Universal Robots URScript: golden_headless.script

# UR5 - Protocole etalement cosmetique
# Genere automatiquement par ur5_etalement.py
# IMPORTANT : calibrer ROBOT_X_ORIGIN, ROBOT_Y_ORIGIN, ROBOT_Z_SURFACE avant execution
#
# === RECETTE DE REPRODUCTION ===
# Ce bloc enonce ce qui a produit ce fichier. Il ne porte pas de date :
# une date rendrait l export non reproductible, et git la porte deja.
# cycles : 6
#   cycle 1 : type=circular waypoints=83    label=Cycle 1 - Circulaire (0deg)
#   cycle 2 : type=circular waypoints=83    label=Cycle 2 - Circulaire (90deg)
#   cycle 3 : type=circular waypoints=83    label=Cycle 3 - Circulaire (0deg)
#   cycle 4 : type=linear   waypoints=26    label=Cycle 4 - Rectiligne (0deg)
#   cycle 5 : type=linear   waypoints=26    label=Cycle 5 - Rectiligne (90deg)
#   cycle 6 : type=linear   waypoints=26    label=Cycle 6 - Rectiligne (0deg)
# empreinte des reglages : 44136fa
#
# === PINCE 2F-85 : AUCUN ACTIONNEMENT ===
# Ce programme n a pas de commande de pince. La 2F-85 est un support
# passif pour le doigt silicone ; seule sa longueur (TCP_GRIPPER_Z=145 mm)
# entre dans set_tcp(). Aucun rq_activate / rq_* / RS485 outil / set_payload.
# Erreur PolyScope "wait for activation completed" au chargement = URCap
# Robotiq Grippers de l INSTALLATION du robot (auto-activation BeforeStart),
# pas ce fichier. Corriger sur le robot : Installation > URCaps/Gripper >
# desactiver l auto-activation, ou retirer le URCap, ou charger sur une
# installation sans pince.
#

# --- Ancre de la zone d'etalement ---
global P_REF = p[-0.011, 0.6, 0.05, 3.14159, 0.0, 0.0]

# --- Vitesses (m/s) par phase ---
# Note : URSCRIPT_MAX_TCP_SPEED (limite PolyScope, 0.25 m/s) n'est pas
# emis ici ; il est applique par le controleur. La vitesse de transit
# est inlinee directement sur les movel de transit.
global URSCRIPT_CONTACT_V = 0.0500  #sym:URSCRIPT_CONTACT_V
global URSCRIPT_RECONTACT_V = 0.0100  #sym:URSCRIPT_RECONTACT_V
global V_CIRC = 0.0360  #sym:CIRC_SPEED
global V_RECT = 0.0800  #sym:LIN_SPEED

# --- Accelerations (m/s^2) par phase ---
global URSCRIPT_ACCEL = 0.8  #sym:URSCRIPT_ACCEL
global A_INIT = 1.2  #sym:A_INIT

# --- Facteurs multiplicateurs globaux ---
global SPEED_FACTOR = 1.0
global ACCEL_FACTOR = 1.0
global URSCRIPT_BLEND = 0.002  #sym:URSCRIPT_BLEND

# --- Sondage de surface : 1 point en Z (sondage 3 points DESACTIVE, voir bloc commente) ---
global PROBE_FORCE_THR    = 4.0
global PROBE_DESCENT_V    = 0.0040
global PROBE_ACCEL        = 0.05
global PROBE_MAX_TRAVEL   = 0.15
global NOMINAL_FRAME = p[-0.011000, 0.592930, 0.050004, 3.141576, 0.000000, 0.000000]
global MEAS_FRAME = p[-0.011000, 0.592930, 0.050004, 3.141576, 0.000000, 0.000000]
global contact_found = False
global contact_pose = p[0,0,0,0,0,0]

# --- Sondage Z (1 point) : trouve le plan de la plaque par contact force ---
# Depart = pose courante (operateur jogge le doigt juste au-dessus du
# plateau). Descente en -Z (base) jusqu au contact ; le Z touche devient
# la reference de TOUS les cycles 1 a 6 via MEAS_FRAME.
def probe_surface_z():
  textmsg(">>> Sondage Z : 1 point (recherche du plateau)")
  start_pose = get_actual_tcp_pose()
  zero_ftsensor()
  sleep(0.2)
  # CB3 (PolyScope 3.x) : descente surveillee dans le thread principal
  # (speedl non bloquant + lecture force + stopl). Pas de thread (stopl/
  # movel interdits dans un thread). get_tcp_force() lu en entier, norme
  # calculee a la main (pas de slice [0:3], absent du parser CB3).
  f_norm = 0.0
  travel = 0.0
  while f_norm <= PROBE_FORCE_THR and travel < PROBE_MAX_TRAVEL:
    speedl([0, 0, -PROBE_DESCENT_V, 0, 0, 0], PROBE_ACCEL, 0.05)
    F_tcp = get_tcp_force()
    f_norm = sqrt(F_tcp[0]*F_tcp[0] + F_tcp[1]*F_tcp[1] + F_tcp[2]*F_tcp[2])
    cur = get_actual_tcp_pose()
    travel = start_pose[2] - cur[2]
  end
  stopl(2.0)
  if f_norm <= PROBE_FORCE_THR:
    popup("Sondage Z echoue - aucun contact", "Rapprocher le doigt du plateau puis relancer", error=True)
    halt
  end
  touch = get_actual_tcp_pose()
  # Reference Z des cycles : repere nominal translate en Z jusqu au plan
  # touche. Orientation/XY restent nominaux (1 point ne mesure pas
  # l inclinaison -> rework futur). apply_correction decale chaque
  # waypoint du meme dz ; force_mode(MEAS_FRAME) regule les 6 N en Z.
  MEAS_FRAME = p[NOMINAL_FRAME[0], NOMINAL_FRAME[1], touch[2], NOMINAL_FRAME[3], NOMINAL_FRAME[4], NOMINAL_FRAME[5]]
  textmsg("Plateau detecte, Z (m) = ", touch[2])
end

def apply_correction(p_world):
  return pose_trans(MEAS_FRAME, pose_trans(pose_inv(NOMINAL_FRAME), p_world))
end

def cycle_1():
  # --- Cycle 1 - Circulaire (0deg) ---
  movel(apply_correction(p[-0.017788, 0.586142, 0.060004, 3.141576, 0.000000, 0.000000]), a=URSCRIPT_ACCEL*ACCEL_FACTOR, v=0.2500*SPEED_FACTOR)
  sleep(0.2)
  zero_ftsensor()
  sleep(0.2)
  force_mode(MEAS_FRAME, [0, 0, 1, 0, 0, 0], [0, 0, -6.0, 0, 0, 0], 2, [0.008, 0.008, 0.04, 0.35, 0.35, 0.35])
  movel(apply_correction(p[-0.017788, 0.586142, 0.045004, 3.141576, 0.000000, 0.000000]), a=URSCRIPT_ACCEL*ACCEL_FACTOR, v=URSCRIPT_RECONTACT_V*SPEED_FACTOR)
  movel(apply_correction(p[-0.017788, 0.586142, 0.050004, 3.141576, 0.000000, 0.000000]), a=URSCRIPT_ACCEL*ACCEL_FACTOR, v=V_CIRC*SPEED_FACTOR, r=URSCRIPT_BLEND)
  movel(apply_correction(p[-0.005291, 0.586502, 0.050004, 3.141576, 0.000000, 0.000000]), a=URSCRIPT_ACCEL*ACCEL_FACTOR, v=V_CIRC*SPEED_FACTOR, r=URSCRIPT_BLEND)
  movel(apply_correction(p[-0.008415, 0.596171, 0.050004, 3.141576, 0.000000, 0.000000]), a=URSCRIPT_ACCEL*ACCEL_FACTOR, v=V_CIRC*SPEED_FACTOR, r=URSCRIPT_BLEND)
  movel(apply_correction(p[-0.016727, 0.588412, 0.050004, 3.141576, 0.000000, 0.000000]), a=URSCRIPT_ACCEL*ACCEL_FACTOR, v=V_CIRC*SPEED_FACTOR, r=URSCRIPT_BLEND)
  movel(apply_correction(p[-0.006870, 0.579901, 0.050004, 3.141576, 0.000000, 0.000000]), a=URSCRIPT_ACCEL*ACCEL_FACTOR, v=V_CIRC*SPEED_FACTOR, r=URSCRIPT_BLEND)
  movel(apply_correction(p[-0.000746, 0.589189, 0.050004, 3.141576, 0.000000, 0.000000]), a=URSCRIPT_ACCEL*ACCEL_FACTOR, v=V_CIRC*SPEED_FACTOR, r=URSCRIPT_BLEND)
  movel(apply_correction(p[-0.010687, 0.590761, 0.050004, 3.141576, 0.000000, 0.000000]), a=URSCRIPT_ACCEL*ACCEL_FACTOR, v=V_CIRC*SPEED_FACTOR, r=URSCRIPT_BLEND)
  movel(apply_correction(p[-0.009818, 0.578226, 0.050004, 3.141576, 0.000000, 0.000000]), a=URSCRIPT_ACCEL*ACCEL_FACTOR, v=V_CIRC*SPEED_FACTOR, r=URSCRIPT_BLEND)
  movel(apply_correction(p[0.002437, 0.579691, 0.050004, 3.141576, 0.000000, 0.000000]), a=URSCRIPT_ACCEL*ACCEL_FACTOR, v=V_CIRC*SPEED_FACTOR, r=URSCRIPT_BLEND)
  movel(apply_correction(p[-0.001599, 0.588917, 0.050004, 3.141576, 0.000000, 0.000000]), a=URSCRIPT_ACCEL*ACCEL_FACTOR, v=V_CIRC*SPEED_FACTOR, r=URSCRIPT_BLEND)
  movel(apply_correction(p[-0.009333, 0.580482, 0.050004, 3.141576, 0.000000, 0.000000]), a=URSCRIPT_ACCEL*ACCEL_FACTOR, v=V_CIRC*SPEED_FACTOR, r=URSCRIPT_BLEND)
  movel(apply_correction(p[0.000969, 0.572620, 0.050004, 3.141576, 0.000000, 0.000000]), a=URSCRIPT_ACCEL*ACCEL_FACTOR, v=V_CIRC*SPEED_FACTOR, r=URSCRIPT_BLEND)
  movel(apply_correction(p[0.006458, 0.582148, 0.050004, 3.141576, 0.000000, 0.000000]), a=URSCRIPT_ACCEL*ACCEL_FACTOR, v=V_CIRC*SPEED_FACTOR, r=URSCRIPT_BLEND)
  movel(apply_correction(p[-0.003817, 0.582897, 0.050004, 3.141576, 0.000000, 0.000000]), a=URSCRIPT_ACCEL*ACCEL_FACTOR, v=V_CIRC*SPEED_FACTOR, r=URSCRIPT_BLEND)
  movel(apply_correction(p[-0.001841, 0.570398, 0.050004, 3.141576, 0.000000, 0.000000]), a=URSCRIPT_ACCEL*ACCEL_FACTOR, v=V_CIRC*SPEED_FACTOR, r=URSCRIPT_BLEND)
  movel(apply_correction(p[0.010119, 0.572931, 0.050004, 3.141576, 0.000000, 0.000000]), a=URSCRIPT_ACCEL*ACCEL_FACTOR, v=V_CIRC*SPEED_FACTOR, r=URSCRIPT_BLEND)
  movel(apply_correction(p[0.005116, 0.581618, 0.050004, 3.141576, 0.000000, 0.000000]), a=URSCRIPT_ACCEL*ACCEL_FACTOR, v=V_CIRC*SPEED_FACTOR, r=URSCRIPT_BLEND)
  movel(apply_correction(p[-0.001866, 0.572369, 0.050004, 3.141576, 0.000000, 0.000000]), a=URSCRIPT_ACCEL*ACCEL_FACTOR, v=V_CIRC*SPEED_FACTOR, r=URSCRIPT_BLEND)
  movel(apply_correction(p[0.009049, 0.565429, 0.050004, 3.141576, 0.000000, 0.000000]), a=URSCRIPT_ACCEL*ACCEL_FACTOR, v=V_CIRC*SPEED_FACTOR, r=URSCRIPT_BLEND)
  movel(apply_correction(p[0.013497, 0.575336, 0.050004, 3.141576, 0.000000, 0.000000]), a=URSCRIPT_ACCEL*ACCEL_FACTOR, v=V_CIRC*SPEED_FACTOR, r=URSCRIPT_BLEND)
  movel(apply_correction(p[0.003100, 0.574984, 0.050004, 3.141576, 0.000000, 0.000000]), a=URSCRIPT_ACCEL*ACCEL_FACTOR, v=V_CIRC*SPEED_FACTOR, r=URSCRIPT_BLEND)
  movel(apply_correction(p[0.006175, 0.562627, 0.050005, 3.141576, 0.000000, 0.000000]), a=URSCRIPT_ACCEL*ACCEL_FACTOR, v=V_CIRC*SPEED_FACTOR, r=URSCRIPT_BLEND)
  movel(apply_correction(p[0.011479, 0.556739, 0.050005, 3.141576, 0.000000, 0.000000]), a=URSCRIPT_ACCEL*ACCEL_FACTOR, v=V_CIRC*SPEED_FACTOR, r=URSCRIPT_BLEND)
  movel(apply_correction(p[0.012647, 0.563823, 0.050005, 3.141576, 0.000000, 0.000000]), a=URSCRIPT_ACCEL*ACCEL_FACTOR, v=V_CIRC*SPEED_FACTOR, r=URSCRIPT_BLEND)
  movel(apply_correction(p[-0.002304, 0.566873, 0.050004, 3.141576, 0.000000, 0.000000]), a=URSCRIPT_ACCEL*ACCEL_FACTOR, v=V_CIRC*SPEED_FACTOR, r=URSCRIPT_BLEND)
  movel(apply_correction(p[-0.004889, 0.556556, 0.050005, 3.141576, 0.000000, 0.000000]), a=URSCRIPT_ACCEL*ACCEL_FACTOR, v=V_CIRC*SPEED_FACTOR, r=URSCRIPT_BLEND)
  movel(apply_correction(p[0.005466, 0.558816, 0.050005, 3.141576, 0.000000, 0.000000]), a=URSCRIPT_ACCEL*ACCEL_FACTOR, v=V_CIRC*SPEED_FACTOR, r=URSCRIPT_BLEND)
  movel(apply_correction(p[0.000547, 0.570683, 0.050004, 3.141576, 0.000000, 0.000000]), a=URSCRIPT_ACCEL*ACCEL_FACTOR, v=V_CIRC*SPEED_FACTOR, r=URSCRIPT_BLEND)
  movel(apply_correction(p[-0.010103, 0.565440, 0.050004, 3.141576, 0.000000, 0.000000]), a=URSCRIPT_ACCEL*ACCEL_FACTOR, v=V_CIRC*SPEED_FACTOR, r=URSCRIPT_BLEND)
  movel(apply_correction(p[-0.002776, 0.558664, 0.050005, 3.141576, 0.000000, 0.000000]), a=URSCRIPT_ACCEL*ACCEL_FACTOR, v=V_CIRC*SPEED_FACTOR, r=URSCRIPT_BLEND)
  movel(apply_correction(p[0.001801, 0.569721, 0.050004, 3.141576, 0.000000, 0.000000]), a=URSCRIPT_ACCEL*ACCEL_FACTOR, v=V_CIRC*SPEED_FACTOR, r=URSCRIPT_BLEND)
  movel(apply_correction(p[-0.010303, 0.573897, 0.050004, 3.141576, 0.000000, 0.000000]), a=URSCRIPT_ACCEL*ACCEL_FACTOR, v=V_CIRC*SPEED_FACTOR, r=URSCRIPT_BLEND)
  movel(apply_correction(p[-0.011785, 0.563486, 0.050005, 3.141576, 0.000000, 0.000000]), a=URSCRIPT_ACCEL*ACCEL_FACTOR, v=V_CIRC*SPEED_FACTOR, r=URSCRIPT_BLEND)
  movel(apply_correction(p[-0.001599, 0.566840, 0.050004, 3.141576, 0.000000, 0.000000]), a=URSCRIPT_ACCEL*ACCEL_FACTOR, v=V_CIRC*SPEED_FACTOR, r=URSCRIPT_BLEND)
  movel(apply_correction(p[-0.007541, 0.578284, 0.050004, 3.141576, 0.000000, 0.000000]), a=URSCRIPT_ACCEL*ACCEL_FACTOR, v=V_CIRC*SPEED_FACTOR, r=URSCRIPT_BLEND)
  movel(apply_correction(p[-0.017540, 0.572147, 0.050004, 3.141576, 0.000000, 0.000000]), a=URSCRIPT_ACCEL*ACCEL_FACTOR, v=V_CIRC*SPEED_FACTOR, r=URSCRIPT_BLEND)
  movel(apply_correction(p[-0.009497, 0.566215, 0.050004, 3.141576, 0.000000, 0.000000]), a=URSCRIPT_ACCEL*ACCEL_FACTOR, v=V_CIRC*SPEED_FACTOR, r=URSCRIPT_BLEND)
  movel(apply_correction(p[-0.005910, 0.577769, 0.050004, 3.141576, 0.000000, 0.000000]), a=URSCRIPT_ACCEL*ACCEL_FACTOR, v=V_CIRC*SPEED_FACTOR, r=URSCRIPT_BLEND)
  movel(apply_correction(p[-0.018263, 0.580865, 0.050004, 3.141576, 0.000000, 0.000000]), a=URSCRIPT_ACCEL*ACCEL_FACTOR, v=V_CIRC*SPEED_FACTOR, r=URSCRIPT_BLEND)
  movel(apply_correction(p[-0.018637, 0.570467, 0.050004, 3.141576, 0.000000, 0.000000]), a=URSCRIPT_ACCEL*ACCEL_FACTOR, v=V_CIRC*SPEED_FACTOR, r=URSCRIPT_BLEND)
  movel(apply_correction(p[-0.018159, 0.585624, 0.050004, 3.141576, 0.000000, 0.000000]), a=URSCRIPT_ACCEL*ACCEL_FACTOR, v=V_CIRC*SPEED_FACTOR, r=URSCRIPT_BLEND)
  movel(apply_correction(p[-0.028128, 0.571383, 0.050004, 3.141576, 0.000000, 0.000000]), a=URSCRIPT_ACCEL*ACCEL_FACTOR, v=V_CIRC*SPEED_FACTOR, r=URSCRIPT_BLEND)
  movel(apply_correction(p[-0.017409, 0.571005, 0.050004, 3.141576, 0.000000, 0.000000]), a=URSCRIPT_ACCEL*ACCEL_FACTOR, v=V_CIRC*SPEED_FACTOR, r=URSCRIPT_BLEND)
  movel(apply_correction(p[-0.028584, 0.563651, 0.050005, 3.141576, 0.000000, 0.000000]), a=URSCRIPT_ACCEL*ACCEL_FACTOR, v=V_CIRC*SPEED_FACTOR, r=URSCRIPT_BLEND)
  movel(apply_correction(p[-0.016049, 0.562454, 0.050005, 3.141576, 0.000000, 0.000000]), a=URSCRIPT_ACCEL*ACCEL_FACTOR, v=V_CIRC*SPEED_FACTOR, r=URSCRIPT_BLEND)
  movel(apply_correction(p[-0.017564, 0.572580, 0.050004, 3.141576, 0.000000, 0.000000]), a=URSCRIPT_ACCEL*ACCEL_FACTOR, v=V_CIRC*SPEED_FACTOR, r=URSCRIPT_BLEND)
  movel(apply_correction(p[-0.026767, 0.566382, 0.050004, 3.141576, 0.000000, 0.000000]), a=URSCRIPT_ACCEL*ACCEL_FACTOR, v=V_CIRC*SPEED_FACTOR, r=URSCRIPT_BLEND)
  movel(apply_correction(p[-0.018293, 0.556563, 0.050005, 3.141576, 0.000000, 0.000000]), a=URSCRIPT_ACCEL*ACCEL_FACTOR, v=V_CIRC*SPEED_FACTOR, r=URSCRIPT_BLEND)
  movel(apply_correction(p[-0.010472, 0.564778, 0.050005, 3.141576, 0.000000, 0.000000]), a=URSCRIPT_ACCEL*ACCEL_FACTOR, v=V_CIRC*SPEED_FACTOR, r=URSCRIPT_BLEND)
  movel(apply_correction(p[-0.020020, 0.568103, 0.050004, 3.141576, 0.000000, 0.000000]), a=URSCRIPT_ACCEL*ACCEL_FACTOR, v=V_CIRC*SPEED_FACTOR, r=URSCRIPT_BLEND)
  movel(apply_correction(p[-0.020718, 0.555702, 0.050005, 3.141576, 0.000000, 0.000000]), a=URSCRIPT_ACCEL*ACCEL_FACTOR, v=V_CIRC*SPEED_FACTOR, r=URSCRIPT_BLEND)
  movel(apply_correction(p[-0.008223, 0.555612, 0.050005, 3.141576, 0.000000, 0.000000]), a=URSCRIPT_ACCEL*ACCEL_FACTOR, v=V_CIRC*SPEED_FACTOR, r=URSCRIPT_BLEND)
  movel(apply_correction(p[-0.010804, 0.565438, 0.050004, 3.141576, 0.000000, 0.000000]), a=URSCRIPT_ACCEL*ACCEL_FACTOR, v=V_CIRC*SPEED_FACTOR, r=URSCRIPT_BLEND)
  movel(apply_correction(p[-0.019465, 0.558275, 0.050005, 3.141576, 0.000000, 0.000000]), a=URSCRIPT_ACCEL*ACCEL_FACTOR, v=V_CIRC*SPEED_FACTOR, r=URSCRIPT_BLEND)
  movel(apply_correction(p[-0.010180, 0.549212, 0.050005, 3.141576, 0.000000, 0.000000]), a=URSCRIPT_ACCEL*ACCEL_FACTOR, v=V_CIRC*SPEED_FACTOR, r=URSCRIPT_BLEND)
  movel(apply_correction(p[-0.003284, 0.558036, 0.050005, 3.141576, 0.000000, 0.000000]), a=URSCRIPT_ACCEL*ACCEL_FACTOR, v=V_CIRC*SPEED_FACTOR, r=URSCRIPT_BLEND)
  movel(apply_correction(p[-0.013205, 0.560317, 0.050005, 3.141576, 0.000000, 0.000000]), a=URSCRIPT_ACCEL*ACCEL_FACTOR, v=V_CIRC*SPEED_FACTOR, r=URSCRIPT_BLEND)
  movel(apply_correction(p[-0.012803, 0.547801, 0.050005, 3.141576, 0.000000, 0.000000]), a=URSCRIPT_ACCEL*ACCEL_FACTOR, v=V_CIRC*SPEED_FACTOR, r=URSCRIPT_BLEND)
  movel(apply_correction(p[-0.000454, 0.548808, 0.050005, 3.141576, 0.000000, 0.000000]), a=URSCRIPT_ACCEL*ACCEL_FACTOR, v=V_CIRC*SPEED_FACTOR, r=URSCRIPT_BLEND)
  movel(apply_correction(p[-0.001819, 0.552639, 0.050005, 3.141576, 0.000000, 0.000000]), a=URSCRIPT_ACCEL*ACCEL_FACTOR, v=V_CIRC*SPEED_FACTOR, r=URSCRIPT_BLEND)
  movel(apply_correction(p[-0.017675, 0.540361, 0.050005, 3.141576, 0.000000, 0.000000]), a=URSCRIPT_ACCEL*ACCEL_FACTOR, v=V_CIRC*SPEED_FACTOR, r=URSCRIPT_BLEND)
  movel(apply_correction(p[-0.021722, 0.540328, 0.050005, 3.141576, 0.000000, 0.000000]), a=URSCRIPT_ACCEL*ACCEL_FACTOR, v=V_CIRC*SPEED_FACTOR, r=URSCRIPT_BLEND)
  movel(apply_correction(p[-0.011399, 0.539911, 0.050005, 3.141576, 0.000000, 0.000000]), a=URSCRIPT_ACCEL*ACCEL_FACTOR, v=V_CIRC*SPEED_FACTOR, r=URSCRIPT_BLEND)
  movel(apply_correction(p[-0.013708, 0.552379, 0.050005, 3.141576, 0.000000, 0.000000]), a=URSCRIPT_ACCEL*ACCEL_FACTOR, v=V_CIRC*SPEED_FACTOR, r=URSCRIPT_BLEND)
  movel(apply_correction(p[-0.025558, 0.549529, 0.050005, 3.141576, 0.000000, 0.000000]), a=URSCRIPT_ACCEL*ACCEL_FACTOR, v=V_CIRC*SPEED_FACTOR, r=URSCRIPT_BLEND)
  movel(apply_correction(p[-0.020274, 0.541023, 0.050005, 3.141576, 0.000000, 0.000000]), a=URSCRIPT_ACCEL*ACCEL_FACTOR, v=V_CIRC*SPEED_FACTOR, r=URSCRIPT_BLEND)
  movel(apply_correction(p[-0.013534, 0.550503, 0.050005, 3.141576, 0.000000, 0.000000]), a=URSCRIPT_ACCEL*ACCEL_FACTOR, v=V_CIRC*SPEED_FACTOR, r=URSCRIPT_BLEND)
  movel(apply_correction(p[-0.024617, 0.557152, 0.050005, 3.141576, 0.000000, 0.000000]), a=URSCRIPT_ACCEL*ACCEL_FACTOR, v=V_CIRC*SPEED_FACTOR, r=URSCRIPT_BLEND)
  movel(apply_correction(p[-0.028743, 0.547152, 0.050005, 3.141576, 0.000000, 0.000000]), a=URSCRIPT_ACCEL*ACCEL_FACTOR, v=V_CIRC*SPEED_FACTOR, r=URSCRIPT_BLEND)
  movel(apply_correction(p[-0.018331, 0.547838, 0.050005, 3.141576, 0.000000, 0.000000]), a=URSCRIPT_ACCEL*ACCEL_FACTOR, v=V_CIRC*SPEED_FACTOR, r=URSCRIPT_BLEND)
  movel(apply_correction(p[-0.021734, 0.560131, 0.050005, 3.141576, 0.000000, 0.000000]), a=URSCRIPT_ACCEL*ACCEL_FACTOR, v=V_CIRC*SPEED_FACTOR, r=URSCRIPT_BLEND)
  movel(apply_correction(p[-0.033158, 0.556261, 0.050005, 3.141576, 0.000000, 0.000000]), a=URSCRIPT_ACCEL*ACCEL_FACTOR, v=V_CIRC*SPEED_FACTOR, r=URSCRIPT_BLEND)
  movel(apply_correction(p[-0.026980, 0.548411, 0.050005, 3.141576, 0.000000, 0.000000]), a=URSCRIPT_ACCEL*ACCEL_FACTOR, v=V_CIRC*SPEED_FACTOR, r=URSCRIPT_BLEND)
  movel(apply_correction(p[-0.021089, 0.558603, 0.050005, 3.141576, 0.000000, 0.000000]), a=URSCRIPT_ACCEL*ACCEL_FACTOR, v=V_CIRC*SPEED_FACTOR, r=URSCRIPT_BLEND)
  movel(apply_correction(p[-0.032663, 0.564261, 0.050005, 3.141576, 0.000000, 0.000000]), a=URSCRIPT_ACCEL*ACCEL_FACTOR, v=V_CIRC*SPEED_FACTOR, r=URSCRIPT_BLEND)
  movel(apply_correction(p[-0.035709, 0.554015, 0.050005, 3.141576, 0.000000, 0.000000]), a=URSCRIPT_ACCEL*ACCEL_FACTOR, v=V_CIRC*SPEED_FACTOR, r=URSCRIPT_BLEND)
  movel(apply_correction(p[-0.025315, 0.555810, 0.050005, 3.141576, 0.000000, 0.000000]), a=URSCRIPT_ACCEL*ACCEL_FACTOR, v=V_CIRC*SPEED_FACTOR, r=URSCRIPT_BLEND)
  movel(apply_correction(p[-0.029475, 0.567681, 0.050004, 3.141576, 0.000000, 0.000000]), a=URSCRIPT_ACCEL*ACCEL_FACTOR, v=V_CIRC*SPEED_FACTOR, r=URSCRIPT_BLEND)
  movel(apply_correction(p[-0.040636, 0.563198, 0.050005, 3.141576, 0.000000, 0.000000]), a=URSCRIPT_ACCEL*ACCEL_FACTOR, v=V_CIRC*SPEED_FACTOR, r=URSCRIPT_BLEND)
  movel(apply_correction(p[-0.033843, 0.555836, 0.050005, 3.141576, 0.000000, 0.000000]), a=URSCRIPT_ACCEL*ACCEL_FACTOR, v=V_CIRC*SPEED_FACTOR, r=URSCRIPT_BLEND)
  movel(apply_correction(p[-0.028668, 0.566586, 0.050004, 3.141576, 0.000000, 0.000000]), a=URSCRIPT_ACCEL*ACCEL_FACTOR, v=V_CIRC*SPEED_FACTOR, r=URSCRIPT_BLEND)
  movel(apply_correction(p[-0.040654, 0.571321, 0.050004, 3.141576, 0.000000, 0.000000]), a=URSCRIPT_ACCEL*ACCEL_FACTOR, v=V_CIRC*SPEED_FACTOR, r=URSCRIPT_BLEND)
  movel(apply_correction(p[-0.042820, 0.561110, 0.050005, 3.141576, 0.000000, 0.000000]), a=URSCRIPT_ACCEL*ACCEL_FACTOR, v=V_CIRC*SPEED_FACTOR, r=URSCRIPT_BLEND)
  end_force_mode()
  movel(apply_correction(p[-0.042820, 0.561110, 0.060005, 3.141576, 0.000000, 0.000000]), a=URSCRIPT_ACCEL*ACCEL_FACTOR, v=0.2500*SPEED_FACTOR)
end

def cycle_2():
  # --- Cycle 2 - Circulaire (90deg) ---
  movel(apply_correction(p[-0.032496, 0.557857, 0.060005, 3.141576, 0.000000, 0.000000]), a=URSCRIPT_ACCEL*ACCEL_FACTOR, v=0.2500*SPEED_FACTOR)
  sleep(0.2)
  zero_ftsensor()
  sleep(0.2)
  force_mode(MEAS_FRAME, [0, 0, 1, 0, 0, 0], [0, 0, -6.0, 0, 0, 0], 2, [0.008, 0.008, 0.04, 0.35, 0.35, 0.35])
  movel(apply_correction(p[-0.032496, 0.557857, 0.045005, 3.141576, 0.000000, 0.000000]), a=URSCRIPT_ACCEL*ACCEL_FACTOR, v=URSCRIPT_RECONTACT_V*SPEED_FACTOR)
  movel(apply_correction(p[-0.032496, 0.557857, 0.050005, 3.141576, 0.000000, 0.000000]), a=URSCRIPT_ACCEL*ACCEL_FACTOR, v=V_CIRC*SPEED_FACTOR, r=URSCRIPT_BLEND)
  movel(apply_correction(p[-0.032857, 0.570355, 0.050004, 3.141576, 0.000000, 0.000000]), a=URSCRIPT_ACCEL*ACCEL_FACTOR, v=V_CIRC*SPEED_FACTOR, r=URSCRIPT_BLEND)
  movel(apply_correction(p[-0.042526, 0.567231, 0.050004, 3.141576, 0.000000, 0.000000]), a=URSCRIPT_ACCEL*ACCEL_FACTOR, v=V_CIRC*SPEED_FACTOR, r=URSCRIPT_BLEND)
  movel(apply_correction(p[-0.034767, 0.558919, 0.050005, 3.141576, 0.000000, 0.000000]), a=URSCRIPT_ACCEL*ACCEL_FACTOR, v=V_CIRC*SPEED_FACTOR, r=URSCRIPT_BLEND)
  movel(apply_correction(p[-0.026256, 0.568776, 0.050004, 3.141576, 0.000000, 0.000000]), a=URSCRIPT_ACCEL*ACCEL_FACTOR, v=V_CIRC*SPEED_FACTOR, r=URSCRIPT_BLEND)
  movel(apply_correction(p[-0.035543, 0.574899, 0.050004, 3.141576, 0.000000, 0.000000]), a=URSCRIPT_ACCEL*ACCEL_FACTOR, v=V_CIRC*SPEED_FACTOR, r=URSCRIPT_BLEND)
  movel(apply_correction(p[-0.037115, 0.564958, 0.050005, 3.141576, 0.000000, 0.000000]), a=URSCRIPT_ACCEL*ACCEL_FACTOR, v=V_CIRC*SPEED_FACTOR, r=URSCRIPT_BLEND)
  movel(apply_correction(p[-0.024580, 0.565827, 0.050004, 3.141576, 0.000000, 0.000000]), a=URSCRIPT_ACCEL*ACCEL_FACTOR, v=V_CIRC*SPEED_FACTOR, r=URSCRIPT_BLEND)
  movel(apply_correction(p[-0.026045, 0.578083, 0.050004, 3.141576, 0.000000, 0.000000]), a=URSCRIPT_ACCEL*ACCEL_FACTOR, v=V_CIRC*SPEED_FACTOR, r=URSCRIPT_BLEND)
  movel(apply_correction(p[-0.035271, 0.574047, 0.050004, 3.141576, 0.000000, 0.000000]), a=URSCRIPT_ACCEL*ACCEL_FACTOR, v=V_CIRC*SPEED_FACTOR, r=URSCRIPT_BLEND)
  movel(apply_correction(p[-0.026836, 0.566313, 0.050004, 3.141576, 0.000000, 0.000000]), a=URSCRIPT_ACCEL*ACCEL_FACTOR, v=V_CIRC*SPEED_FACTOR, r=URSCRIPT_BLEND)
  movel(apply_correction(p[-0.018974, 0.576615, 0.050004, 3.141576, 0.000000, 0.000000]), a=URSCRIPT_ACCEL*ACCEL_FACTOR, v=V_CIRC*SPEED_FACTOR, r=URSCRIPT_BLEND)
  movel(apply_correction(p[-0.028502, 0.582104, 0.050004, 3.141576, 0.000000, 0.000000]), a=URSCRIPT_ACCEL*ACCEL_FACTOR, v=V_CIRC*SPEED_FACTOR, r=URSCRIPT_BLEND)
  movel(apply_correction(p[-0.029251, 0.571829, 0.050004, 3.141576, 0.000000, 0.000000]), a=URSCRIPT_ACCEL*ACCEL_FACTOR, v=V_CIRC*SPEED_FACTOR, r=URSCRIPT_BLEND)
  movel(apply_correction(p[-0.016752, 0.573805, 0.050004, 3.141576, 0.000000, 0.000000]), a=URSCRIPT_ACCEL*ACCEL_FACTOR, v=V_CIRC*SPEED_FACTOR, r=URSCRIPT_BLEND)
  movel(apply_correction(p[-0.019285, 0.585765, 0.050004, 3.141576, 0.000000, 0.000000]), a=URSCRIPT_ACCEL*ACCEL_FACTOR, v=V_CIRC*SPEED_FACTOR, r=URSCRIPT_BLEND)
  movel(apply_correction(p[-0.027972, 0.580762, 0.050004, 3.141576, 0.000000, 0.000000]), a=URSCRIPT_ACCEL*ACCEL_FACTOR, v=V_CIRC*SPEED_FACTOR, r=URSCRIPT_BLEND)
  movel(apply_correction(p[-0.018723, 0.573780, 0.050004, 3.141576, 0.000000, 0.000000]), a=URSCRIPT_ACCEL*ACCEL_FACTOR, v=V_CIRC*SPEED_FACTOR, r=URSCRIPT_BLEND)
  movel(apply_correction(p[-0.011783, 0.584695, 0.050004, 3.141576, 0.000000, 0.000000]), a=URSCRIPT_ACCEL*ACCEL_FACTOR, v=V_CIRC*SPEED_FACTOR, r=URSCRIPT_BLEND)
  movel(apply_correction(p[-0.021690, 0.589143, 0.050004, 3.141576, 0.000000, 0.000000]), a=URSCRIPT_ACCEL*ACCEL_FACTOR, v=V_CIRC*SPEED_FACTOR, r=URSCRIPT_BLEND)
  movel(apply_correction(p[-0.021339, 0.578746, 0.050004, 3.141576, 0.000000, 0.000000]), a=URSCRIPT_ACCEL*ACCEL_FACTOR, v=V_CIRC*SPEED_FACTOR, r=URSCRIPT_BLEND)
  movel(apply_correction(p[-0.008981, 0.581821, 0.050004, 3.141576, 0.000000, 0.000000]), a=URSCRIPT_ACCEL*ACCEL_FACTOR, v=V_CIRC*SPEED_FACTOR, r=URSCRIPT_BLEND)
  movel(apply_correction(p[-0.003093, 0.587125, 0.050004, 3.141576, 0.000000, 0.000000]), a=URSCRIPT_ACCEL*ACCEL_FACTOR, v=V_CIRC*SPEED_FACTOR, r=URSCRIPT_BLEND)
  movel(apply_correction(p[-0.010177, 0.588293, 0.050004, 3.141576, 0.000000, 0.000000]), a=URSCRIPT_ACCEL*ACCEL_FACTOR, v=V_CIRC*SPEED_FACTOR, r=URSCRIPT_BLEND)
  movel(apply_correction(p[-0.013227, 0.573342, 0.050004, 3.141576, 0.000000, 0.000000]), a=URSCRIPT_ACCEL*ACCEL_FACTOR, v=V_CIRC*SPEED_FACTOR, r=URSCRIPT_BLEND)
  movel(apply_correction(p[-0.002911, 0.570756, 0.050004, 3.141576, 0.000000, 0.000000]), a=URSCRIPT_ACCEL*ACCEL_FACTOR, v=V_CIRC*SPEED_FACTOR, r=URSCRIPT_BLEND)
  movel(apply_correction(p[-0.005170, 0.581112, 0.050004, 3.141576, 0.000000, 0.000000]), a=URSCRIPT_ACCEL*ACCEL_FACTOR, v=V_CIRC*SPEED_FACTOR, r=URSCRIPT_BLEND)
  movel(apply_correction(p[-0.017037, 0.576193, 0.050004, 3.141576, 0.000000, 0.000000]), a=URSCRIPT_ACCEL*ACCEL_FACTOR, v=V_CIRC*SPEED_FACTOR, r=URSCRIPT_BLEND)
  movel(apply_correction(p[-0.011795, 0.565542, 0.050004, 3.141576, 0.000000, 0.000000]), a=URSCRIPT_ACCEL*ACCEL_FACTOR, v=V_CIRC*SPEED_FACTOR, r=URSCRIPT_BLEND)
  movel(apply_correction(p[-0.005019, 0.572870, 0.050004, 3.141576, 0.000000, 0.000000]), a=URSCRIPT_ACCEL*ACCEL_FACTOR, v=V_CIRC*SPEED_FACTOR, r=URSCRIPT_BLEND)
  movel(apply_correction(p[-0.016075, 0.577446, 0.050004, 3.141576, 0.000000, 0.000000]), a=URSCRIPT_ACCEL*ACCEL_FACTOR, v=V_CIRC*SPEED_FACTOR, r=URSCRIPT_BLEND)
  movel(apply_correction(p[-0.020251, 0.565342, 0.050005, 3.141576, 0.000000, 0.000000]), a=URSCRIPT_ACCEL*ACCEL_FACTOR, v=V_CIRC*SPEED_FACTOR, r=URSCRIPT_BLEND)
  movel(apply_correction(p[-0.009840, 0.563861, 0.050005, 3.141576, 0.000000, 0.000000]), a=URSCRIPT_ACCEL*ACCEL_FACTOR, v=V_CIRC*SPEED_FACTOR, r=URSCRIPT_BLEND)
  movel(apply_correction(p[-0.013194, 0.574047, 0.050004, 3.141576, 0.000000, 0.000000]), a=URSCRIPT_ACCEL*ACCEL_FACTOR, v=V_CIRC*SPEED_FACTOR, r=URSCRIPT_BLEND)
  movel(apply_correction(p[-0.024639, 0.568105, 0.050004, 3.141576, 0.000000, 0.000000]), a=URSCRIPT_ACCEL*ACCEL_FACTOR, v=V_CIRC*SPEED_FACTOR, r=URSCRIPT_BLEND)
  movel(apply_correction(p[-0.018502, 0.558106, 0.050005, 3.141576, 0.000000, 0.000000]), a=URSCRIPT_ACCEL*ACCEL_FACTOR, v=V_CIRC*SPEED_FACTOR, r=URSCRIPT_BLEND)
  movel(apply_correction(p[-0.012570, 0.566149, 0.050004, 3.141576, 0.000000, 0.000000]), a=URSCRIPT_ACCEL*ACCEL_FACTOR, v=V_CIRC*SPEED_FACTOR, r=URSCRIPT_BLEND)
  movel(apply_correction(p[-0.024123, 0.569736, 0.050004, 3.141576, 0.000000, 0.000000]), a=URSCRIPT_ACCEL*ACCEL_FACTOR, v=V_CIRC*SPEED_FACTOR, r=URSCRIPT_BLEND)
  movel(apply_correction(p[-0.027220, 0.557382, 0.050005, 3.141576, 0.000000, 0.000000]), a=URSCRIPT_ACCEL*ACCEL_FACTOR, v=V_CIRC*SPEED_FACTOR, r=URSCRIPT_BLEND)
  movel(apply_correction(p[-0.016822, 0.557008, 0.050005, 3.141576, 0.000000, 0.000000]), a=URSCRIPT_ACCEL*ACCEL_FACTOR, v=V_CIRC*SPEED_FACTOR, r=URSCRIPT_BLEND)
  movel(apply_correction(p[-0.031978, 0.557487, 0.050005, 3.141576, 0.000000, 0.000000]), a=URSCRIPT_ACCEL*ACCEL_FACTOR, v=V_CIRC*SPEED_FACTOR, r=URSCRIPT_BLEND)
  movel(apply_correction(p[-0.017737, 0.547518, 0.050005, 3.141576, 0.000000, 0.000000]), a=URSCRIPT_ACCEL*ACCEL_FACTOR, v=V_CIRC*SPEED_FACTOR, r=URSCRIPT_BLEND)
  movel(apply_correction(p[-0.017359, 0.558237, 0.050005, 3.141576, 0.000000, 0.000000]), a=URSCRIPT_ACCEL*ACCEL_FACTOR, v=V_CIRC*SPEED_FACTOR, r=URSCRIPT_BLEND)
  movel(apply_correction(p[-0.010005, 0.547062, 0.050005, 3.141576, 0.000000, 0.000000]), a=URSCRIPT_ACCEL*ACCEL_FACTOR, v=V_CIRC*SPEED_FACTOR, r=URSCRIPT_BLEND)
  movel(apply_correction(p[-0.008808, 0.559597, 0.050005, 3.141576, 0.000000, 0.000000]), a=URSCRIPT_ACCEL*ACCEL_FACTOR, v=V_CIRC*SPEED_FACTOR, r=URSCRIPT_BLEND)
  movel(apply_correction(p[-0.018934, 0.558082, 0.050005, 3.141576, 0.000000, 0.000000]), a=URSCRIPT_ACCEL*ACCEL_FACTOR, v=V_CIRC*SPEED_FACTOR, r=URSCRIPT_BLEND)
  movel(apply_correction(p[-0.012737, 0.548879, 0.050005, 3.141576, 0.000000, 0.000000]), a=URSCRIPT_ACCEL*ACCEL_FACTOR, v=V_CIRC*SPEED_FACTOR, r=URSCRIPT_BLEND)
  movel(apply_correction(p[-0.002918, 0.557353, 0.050005, 3.141576, 0.000000, 0.000000]), a=URSCRIPT_ACCEL*ACCEL_FACTOR, v=V_CIRC*SPEED_FACTOR, r=URSCRIPT_BLEND)
  movel(apply_correction(p[-0.011132, 0.565174, 0.050005, 3.141576, 0.000000, 0.000000]), a=URSCRIPT_ACCEL*ACCEL_FACTOR, v=V_CIRC*SPEED_FACTOR, r=URSCRIPT_BLEND)
  movel(apply_correction(p[-0.014458, 0.555626, 0.050005, 3.141576, 0.000000, 0.000000]), a=URSCRIPT_ACCEL*ACCEL_FACTOR, v=V_CIRC*SPEED_FACTOR, r=URSCRIPT_BLEND)
  movel(apply_correction(p[-0.002057, 0.554927, 0.050005, 3.141576, 0.000000, 0.000000]), a=URSCRIPT_ACCEL*ACCEL_FACTOR, v=V_CIRC*SPEED_FACTOR, r=URSCRIPT_BLEND)
  movel(apply_correction(p[-0.001967, 0.567422, 0.050004, 3.141576, 0.000000, 0.000000]), a=URSCRIPT_ACCEL*ACCEL_FACTOR, v=V_CIRC*SPEED_FACTOR, r=URSCRIPT_BLEND)
  movel(apply_correction(p[-0.011793, 0.564842, 0.050005, 3.141576, 0.000000, 0.000000]), a=URSCRIPT_ACCEL*ACCEL_FACTOR, v=V_CIRC*SPEED_FACTOR, r=URSCRIPT_BLEND)
  movel(apply_correction(p[-0.004630, 0.556181, 0.050005, 3.141576, 0.000000, 0.000000]), a=URSCRIPT_ACCEL*ACCEL_FACTOR, v=V_CIRC*SPEED_FACTOR, r=URSCRIPT_BLEND)
  movel(apply_correction(p[0.004433, 0.565466, 0.050004, 3.141576, 0.000000, 0.000000]), a=URSCRIPT_ACCEL*ACCEL_FACTOR, v=V_CIRC*SPEED_FACTOR, r=URSCRIPT_BLEND)
  movel(apply_correction(p[-0.004390, 0.572362, 0.050004, 3.141576, 0.000000, 0.000000]), a=URSCRIPT_ACCEL*ACCEL_FACTOR, v=V_CIRC*SPEED_FACTOR, r=URSCRIPT_BLEND)
  movel(apply_correction(p[-0.006672, 0.562440, 0.050005, 3.141576, 0.000000, 0.000000]), a=URSCRIPT_ACCEL*ACCEL_FACTOR, v=V_CIRC*SPEED_FACTOR, r=URSCRIPT_BLEND)
  movel(apply_correction(p[0.005845, 0.562843, 0.050005, 3.141576, 0.000000, 0.000000]), a=URSCRIPT_ACCEL*ACCEL_FACTOR, v=V_CIRC*SPEED_FACTOR, r=URSCRIPT_BLEND)
  movel(apply_correction(p[0.004838, 0.575191, 0.050004, 3.141576, 0.000000, 0.000000]), a=URSCRIPT_ACCEL*ACCEL_FACTOR, v=V_CIRC*SPEED_FACTOR, r=URSCRIPT_BLEND)
  movel(apply_correction(p[0.001007, 0.573827, 0.050004, 3.141576, 0.000000, 0.000000]), a=URSCRIPT_ACCEL*ACCEL_FACTOR, v=V_CIRC*SPEED_FACTOR, r=URSCRIPT_BLEND)
  movel(apply_correction(p[0.013285, 0.557971, 0.050005, 3.141576, 0.000000, 0.000000]), a=URSCRIPT_ACCEL*ACCEL_FACTOR, v=V_CIRC*SPEED_FACTOR, r=URSCRIPT_BLEND)
  movel(apply_correction(p[0.013318, 0.553924, 0.050005, 3.141576, 0.000000, 0.000000]), a=URSCRIPT_ACCEL*ACCEL_FACTOR, v=V_CIRC*SPEED_FACTOR, r=URSCRIPT_BLEND)
  movel(apply_correction(p[0.013735, 0.564247, 0.050005, 3.141576, 0.000000, 0.000000]), a=URSCRIPT_ACCEL*ACCEL_FACTOR, v=V_CIRC*SPEED_FACTOR, r=URSCRIPT_BLEND)
  movel(apply_correction(p[0.001267, 0.561937, 0.050005, 3.141576, 0.000000, 0.000000]), a=URSCRIPT_ACCEL*ACCEL_FACTOR, v=V_CIRC*SPEED_FACTOR, r=URSCRIPT_BLEND)
  movel(apply_correction(p[0.004117, 0.550088, 0.050005, 3.141576, 0.000000, 0.000000]), a=URSCRIPT_ACCEL*ACCEL_FACTOR, v=V_CIRC*SPEED_FACTOR, r=URSCRIPT_BLEND)
  movel(apply_correction(p[0.012622, 0.555372, 0.050005, 3.141576, 0.000000, 0.000000]), a=URSCRIPT_ACCEL*ACCEL_FACTOR, v=V_CIRC*SPEED_FACTOR, r=URSCRIPT_BLEND)
  movel(apply_correction(p[0.003143, 0.562112, 0.050005, 3.141576, 0.000000, 0.000000]), a=URSCRIPT_ACCEL*ACCEL_FACTOR, v=V_CIRC*SPEED_FACTOR, r=URSCRIPT_BLEND)
  movel(apply_correction(p[-0.003507, 0.551029, 0.050005, 3.141576, 0.000000, 0.000000]), a=URSCRIPT_ACCEL*ACCEL_FACTOR, v=V_CIRC*SPEED_FACTOR, r=URSCRIPT_BLEND)
  movel(apply_correction(p[0.006494, 0.546903, 0.050005, 3.141576, 0.000000, 0.000000]), a=URSCRIPT_ACCEL*ACCEL_FACTOR, v=V_CIRC*SPEED_FACTOR, r=URSCRIPT_BLEND)
  movel(apply_correction(p[0.005807, 0.557315, 0.050005, 3.141576, 0.000000, 0.000000]), a=URSCRIPT_ACCEL*ACCEL_FACTOR, v=V_CIRC*SPEED_FACTOR, r=URSCRIPT_BLEND)
  movel(apply_correction(p[-0.006486, 0.553912, 0.050005, 3.141576, 0.000000, 0.000000]), a=URSCRIPT_ACCEL*ACCEL_FACTOR, v=V_CIRC*SPEED_FACTOR, r=URSCRIPT_BLEND)
  movel(apply_correction(p[-0.002615, 0.542488, 0.050005, 3.141576, 0.000000, 0.000000]), a=URSCRIPT_ACCEL*ACCEL_FACTOR, v=V_CIRC*SPEED_FACTOR, r=URSCRIPT_BLEND)
  movel(apply_correction(p[0.005234, 0.548666, 0.050005, 3.141576, 0.000000, 0.000000]), a=URSCRIPT_ACCEL*ACCEL_FACTOR, v=V_CIRC*SPEED_FACTOR, r=URSCRIPT_BLEND)
  movel(apply_correction(p[-0.004957, 0.554557, 0.050005, 3.141576, 0.000000, 0.000000]), a=URSCRIPT_ACCEL*ACCEL_FACTOR, v=V_CIRC*SPEED_FACTOR, r=URSCRIPT_BLEND)
  movel(apply_correction(p[-0.010615, 0.542983, 0.050005, 3.141576, 0.000000, 0.000000]), a=URSCRIPT_ACCEL*ACCEL_FACTOR, v=V_CIRC*SPEED_FACTOR, r=URSCRIPT_BLEND)
  movel(apply_correction(p[-0.000369, 0.539937, 0.050005, 3.141576, 0.000000, 0.000000]), a=URSCRIPT_ACCEL*ACCEL_FACTOR, v=V_CIRC*SPEED_FACTOR, r=URSCRIPT_BLEND)
  movel(apply_correction(p[-0.002164, 0.550331, 0.050005, 3.141576, 0.000000, 0.000000]), a=URSCRIPT_ACCEL*ACCEL_FACTOR, v=V_CIRC*SPEED_FACTOR, r=URSCRIPT_BLEND)
  movel(apply_correction(p[-0.014036, 0.546171, 0.050005, 3.141576, 0.000000, 0.000000]), a=URSCRIPT_ACCEL*ACCEL_FACTOR, v=V_CIRC*SPEED_FACTOR, r=URSCRIPT_BLEND)
  movel(apply_correction(p[-0.009552, 0.535009, 0.050005, 3.141576, 0.000000, 0.000000]), a=URSCRIPT_ACCEL*ACCEL_FACTOR, v=V_CIRC*SPEED_FACTOR, r=URSCRIPT_BLEND)
  movel(apply_correction(p[-0.002190, 0.541803, 0.050005, 3.141576, 0.000000, 0.000000]), a=URSCRIPT_ACCEL*ACCEL_FACTOR, v=V_CIRC*SPEED_FACTOR, r=URSCRIPT_BLEND)
  movel(apply_correction(p[-0.012940, 0.546978, 0.050005, 3.141576, 0.000000, 0.000000]), a=URSCRIPT_ACCEL*ACCEL_FACTOR, v=V_CIRC*SPEED_FACTOR, r=URSCRIPT_BLEND)
  movel(apply_correction(p[-0.017676, 0.534992, 0.050005, 3.141576, 0.000000, 0.000000]), a=URSCRIPT_ACCEL*ACCEL_FACTOR, v=V_CIRC*SPEED_FACTOR, r=URSCRIPT_BLEND)
  movel(apply_correction(p[-0.007464, 0.532826, 0.050005, 3.141576, 0.000000, 0.000000]), a=URSCRIPT_ACCEL*ACCEL_FACTOR, v=V_CIRC*SPEED_FACTOR, r=URSCRIPT_BLEND)
  end_force_mode()
  movel(apply_correction(p[-0.007464, 0.532826, 0.060005, 3.141576, 0.000000, 0.000000]), a=URSCRIPT_ACCEL*ACCEL_FACTOR, v=0.2500*SPEED_FACTOR)
end

def cycle_3():
  # --- Cycle 3 - Circulaire (0deg) ---
  movel(apply_correction(p[-0.017788, 0.586142, 0.060004, 3.141576, 0.000000, 0.000000]), a=URSCRIPT_ACCEL*ACCEL_FACTOR, v=0.2500*SPEED_FACTOR)
  sleep(0.2)
  zero_ftsensor()
  sleep(0.2)
  force_mode(MEAS_FRAME, [0, 0, 1, 0, 0, 0], [0, 0, -6.0, 0, 0, 0], 2, [0.008, 0.008, 0.04, 0.35, 0.35, 0.35])
  movel(apply_correction(p[-0.017788, 0.586142, 0.045004, 3.141576, 0.000000, 0.000000]), a=URSCRIPT_ACCEL*ACCEL_FACTOR, v=URSCRIPT_RECONTACT_V*SPEED_FACTOR)
  movel(apply_correction(p[-0.017788, 0.586142, 0.050004, 3.141576, 0.000000, 0.000000]), a=URSCRIPT_ACCEL*ACCEL_FACTOR, v=V_CIRC*SPEED_FACTOR, r=URSCRIPT_BLEND)
  movel(apply_correction(p[-0.005291, 0.586502, 0.050004, 3.141576, 0.000000, 0.000000]), a=URSCRIPT_ACCEL*ACCEL_FACTOR, v=V_CIRC*SPEED_FACTOR, r=URSCRIPT_BLEND)
  movel(apply_correction(p[-0.008415, 0.596171, 0.050004, 3.141576, 0.000000, 0.000000]), a=URSCRIPT_ACCEL*ACCEL_FACTOR, v=V_CIRC*SPEED_FACTOR, r=URSCRIPT_BLEND)
  movel(apply_correction(p[-0.016727, 0.588412, 0.050004, 3.141576, 0.000000, 0.000000]), a=URSCRIPT_ACCEL*ACCEL_FACTOR, v=V_CIRC*SPEED_FACTOR, r=URSCRIPT_BLEND)
  movel(apply_correction(p[-0.006870, 0.579901, 0.050004, 3.141576, 0.000000, 0.000000]), a=URSCRIPT_ACCEL*ACCEL_FACTOR, v=V_CIRC*SPEED_FACTOR, r=URSCRIPT_BLEND)
  movel(apply_correction(p[-0.000746, 0.589189, 0.050004, 3.141576, 0.000000, 0.000000]), a=URSCRIPT_ACCEL*ACCEL_FACTOR, v=V_CIRC*SPEED_FACTOR, r=URSCRIPT_BLEND)
  movel(apply_correction(p[-0.010687, 0.590761, 0.050004, 3.141576, 0.000000, 0.000000]), a=URSCRIPT_ACCEL*ACCEL_FACTOR, v=V_CIRC*SPEED_FACTOR, r=URSCRIPT_BLEND)
  movel(apply_correction(p[-0.009818, 0.578226, 0.050004, 3.141576, 0.000000, 0.000000]), a=URSCRIPT_ACCEL*ACCEL_FACTOR, v=V_CIRC*SPEED_FACTOR, r=URSCRIPT_BLEND)
  movel(apply_correction(p[0.002437, 0.579691, 0.050004, 3.141576, 0.000000, 0.000000]), a=URSCRIPT_ACCEL*ACCEL_FACTOR, v=V_CIRC*SPEED_FACTOR, r=URSCRIPT_BLEND)
  movel(apply_correction(p[-0.001599, 0.588917, 0.050004, 3.141576, 0.000000, 0.000000]), a=URSCRIPT_ACCEL*ACCEL_FACTOR, v=V_CIRC*SPEED_FACTOR, r=URSCRIPT_BLEND)
  movel(apply_correction(p[-0.009333, 0.580482, 0.050004, 3.141576, 0.000000, 0.000000]), a=URSCRIPT_ACCEL*ACCEL_FACTOR, v=V_CIRC*SPEED_FACTOR, r=URSCRIPT_BLEND)
  movel(apply_correction(p[0.000969, 0.572620, 0.050004, 3.141576, 0.000000, 0.000000]), a=URSCRIPT_ACCEL*ACCEL_FACTOR, v=V_CIRC*SPEED_FACTOR, r=URSCRIPT_BLEND)
  movel(apply_correction(p[0.006458, 0.582148, 0.050004, 3.141576, 0.000000, 0.000000]), a=URSCRIPT_ACCEL*ACCEL_FACTOR, v=V_CIRC*SPEED_FACTOR, r=URSCRIPT_BLEND)
  movel(apply_correction(p[-0.003817, 0.582897, 0.050004, 3.141576, 0.000000, 0.000000]), a=URSCRIPT_ACCEL*ACCEL_FACTOR, v=V_CIRC*SPEED_FACTOR, r=URSCRIPT_BLEND)
  movel(apply_correction(p[-0.001841, 0.570398, 0.050004, 3.141576, 0.000000, 0.000000]), a=URSCRIPT_ACCEL*ACCEL_FACTOR, v=V_CIRC*SPEED_FACTOR, r=URSCRIPT_BLEND)
  movel(apply_correction(p[0.010119, 0.572931, 0.050004, 3.141576, 0.000000, 0.000000]), a=URSCRIPT_ACCEL*ACCEL_FACTOR, v=V_CIRC*SPEED_FACTOR, r=URSCRIPT_BLEND)
  movel(apply_correction(p[0.005116, 0.581618, 0.050004, 3.141576, 0.000000, 0.000000]), a=URSCRIPT_ACCEL*ACCEL_FACTOR, v=V_CIRC*SPEED_FACTOR, r=URSCRIPT_BLEND)
  movel(apply_correction(p[-0.001866, 0.572369, 0.050004, 3.141576, 0.000000, 0.000000]), a=URSCRIPT_ACCEL*ACCEL_FACTOR, v=V_CIRC*SPEED_FACTOR, r=URSCRIPT_BLEND)
  movel(apply_correction(p[0.009049, 0.565429, 0.050004, 3.141576, 0.000000, 0.000000]), a=URSCRIPT_ACCEL*ACCEL_FACTOR, v=V_CIRC*SPEED_FACTOR, r=URSCRIPT_BLEND)
  movel(apply_correction(p[0.013497, 0.575336, 0.050004, 3.141576, 0.000000, 0.000000]), a=URSCRIPT_ACCEL*ACCEL_FACTOR, v=V_CIRC*SPEED_FACTOR, r=URSCRIPT_BLEND)
  movel(apply_correction(p[0.003100, 0.574984, 0.050004, 3.141576, 0.000000, 0.000000]), a=URSCRIPT_ACCEL*ACCEL_FACTOR, v=V_CIRC*SPEED_FACTOR, r=URSCRIPT_BLEND)
  movel(apply_correction(p[0.006175, 0.562627, 0.050005, 3.141576, 0.000000, 0.000000]), a=URSCRIPT_ACCEL*ACCEL_FACTOR, v=V_CIRC*SPEED_FACTOR, r=URSCRIPT_BLEND)
  movel(apply_correction(p[0.011479, 0.556739, 0.050005, 3.141576, 0.000000, 0.000000]), a=URSCRIPT_ACCEL*ACCEL_FACTOR, v=V_CIRC*SPEED_FACTOR, r=URSCRIPT_BLEND)
  movel(apply_correction(p[0.012647, 0.563823, 0.050005, 3.141576, 0.000000, 0.000000]), a=URSCRIPT_ACCEL*ACCEL_FACTOR, v=V_CIRC*SPEED_FACTOR, r=URSCRIPT_BLEND)
  movel(apply_correction(p[-0.002304, 0.566873, 0.050004, 3.141576, 0.000000, 0.000000]), a=URSCRIPT_ACCEL*ACCEL_FACTOR, v=V_CIRC*SPEED_FACTOR, r=URSCRIPT_BLEND)
  movel(apply_correction(p[-0.004889, 0.556556, 0.050005, 3.141576, 0.000000, 0.000000]), a=URSCRIPT_ACCEL*ACCEL_FACTOR, v=V_CIRC*SPEED_FACTOR, r=URSCRIPT_BLEND)
  movel(apply_correction(p[0.005466, 0.558816, 0.050005, 3.141576, 0.000000, 0.000000]), a=URSCRIPT_ACCEL*ACCEL_FACTOR, v=V_CIRC*SPEED_FACTOR, r=URSCRIPT_BLEND)
  movel(apply_correction(p[0.000547, 0.570683, 0.050004, 3.141576, 0.000000, 0.000000]), a=URSCRIPT_ACCEL*ACCEL_FACTOR, v=V_CIRC*SPEED_FACTOR, r=URSCRIPT_BLEND)
  movel(apply_correction(p[-0.010103, 0.565440, 0.050004, 3.141576, 0.000000, 0.000000]), a=URSCRIPT_ACCEL*ACCEL_FACTOR, v=V_CIRC*SPEED_FACTOR, r=URSCRIPT_BLEND)
  movel(apply_correction(p[-0.002776, 0.558664, 0.050005, 3.141576, 0.000000, 0.000000]), a=URSCRIPT_ACCEL*ACCEL_FACTOR, v=V_CIRC*SPEED_FACTOR, r=URSCRIPT_BLEND)
  movel(apply_correction(p[0.001801, 0.569721, 0.050004, 3.141576, 0.000000, 0.000000]), a=URSCRIPT_ACCEL*ACCEL_FACTOR, v=V_CIRC*SPEED_FACTOR, r=URSCRIPT_BLEND)
  movel(apply_correction(p[-0.010303, 0.573897, 0.050004, 3.141576, 0.000000, 0.000000]), a=URSCRIPT_ACCEL*ACCEL_FACTOR, v=V_CIRC*SPEED_FACTOR, r=URSCRIPT_BLEND)
  movel(apply_correction(p[-0.011785, 0.563486, 0.050005, 3.141576, 0.000000, 0.000000]), a=URSCRIPT_ACCEL*ACCEL_FACTOR, v=V_CIRC*SPEED_FACTOR, r=URSCRIPT_BLEND)
  movel(apply_correction(p[-0.001599, 0.566840, 0.050004, 3.141576, 0.000000, 0.000000]), a=URSCRIPT_ACCEL*ACCEL_FACTOR, v=V_CIRC*SPEED_FACTOR, r=URSCRIPT_BLEND)
  movel(apply_correction(p[-0.007541, 0.578284, 0.050004, 3.141576, 0.000000, 0.000000]), a=URSCRIPT_ACCEL*ACCEL_FACTOR, v=V_CIRC*SPEED_FACTOR, r=URSCRIPT_BLEND)
  movel(apply_correction(p[-0.017540, 0.572147, 0.050004, 3.141576, 0.000000, 0.000000]), a=URSCRIPT_ACCEL*ACCEL_FACTOR, v=V_CIRC*SPEED_FACTOR, r=URSCRIPT_BLEND)
  movel(apply_correction(p[-0.009497, 0.566215, 0.050004, 3.141576, 0.000000, 0.000000]), a=URSCRIPT_ACCEL*ACCEL_FACTOR, v=V_CIRC*SPEED_FACTOR, r=URSCRIPT_BLEND)
  movel(apply_correction(p[-0.005910, 0.577769, 0.050004, 3.141576, 0.000000, 0.000000]), a=URSCRIPT_ACCEL*ACCEL_FACTOR, v=V_CIRC*SPEED_FACTOR, r=URSCRIPT_BLEND)
  movel(apply_correction(p[-0.018263, 0.580865, 0.050004, 3.141576, 0.000000, 0.000000]), a=URSCRIPT_ACCEL*ACCEL_FACTOR, v=V_CIRC*SPEED_FACTOR, r=URSCRIPT_BLEND)
  movel(apply_correction(p[-0.018637, 0.570467, 0.050004, 3.141576, 0.000000, 0.000000]), a=URSCRIPT_ACCEL*ACCEL_FACTOR, v=V_CIRC*SPEED_FACTOR, r=URSCRIPT_BLEND)
  movel(apply_correction(p[-0.018159, 0.585624, 0.050004, 3.141576, 0.000000, 0.000000]), a=URSCRIPT_ACCEL*ACCEL_FACTOR, v=V_CIRC*SPEED_FACTOR, r=URSCRIPT_BLEND)
  movel(apply_correction(p[-0.028128, 0.571383, 0.050004, 3.141576, 0.000000, 0.000000]), a=URSCRIPT_ACCEL*ACCEL_FACTOR, v=V_CIRC*SPEED_FACTOR, r=URSCRIPT_BLEND)
  movel(apply_correction(p[-0.017409, 0.571005, 0.050004, 3.141576, 0.000000, 0.000000]), a=URSCRIPT_ACCEL*ACCEL_FACTOR, v=V_CIRC*SPEED_FACTOR, r=URSCRIPT_BLEND)
  movel(apply_correction(p[-0.028584, 0.563651, 0.050005, 3.141576, 0.000000, 0.000000]), a=URSCRIPT_ACCEL*ACCEL_FACTOR, v=V_CIRC*SPEED_FACTOR, r=URSCRIPT_BLEND)
  movel(apply_correction(p[-0.016049, 0.562454, 0.050005, 3.141576, 0.000000, 0.000000]), a=URSCRIPT_ACCEL*ACCEL_FACTOR, v=V_CIRC*SPEED_FACTOR, r=URSCRIPT_BLEND)
  movel(apply_correction(p[-0.017564, 0.572580, 0.050004, 3.141576, 0.000000, 0.000000]), a=URSCRIPT_ACCEL*ACCEL_FACTOR, v=V_CIRC*SPEED_FACTOR, r=URSCRIPT_BLEND)
  movel(apply_correction(p[-0.026767, 0.566382, 0.050004, 3.141576, 0.000000, 0.000000]), a=URSCRIPT_ACCEL*ACCEL_FACTOR, v=V_CIRC*SPEED_FACTOR, r=URSCRIPT_BLEND)
  movel(apply_correction(p[-0.018293, 0.556563, 0.050005, 3.141576, 0.000000, 0.000000]), a=URSCRIPT_ACCEL*ACCEL_FACTOR, v=V_CIRC*SPEED_FACTOR, r=URSCRIPT_BLEND)
  movel(apply_correction(p[-0.010472, 0.564778, 0.050005, 3.141576, 0.000000, 0.000000]), a=URSCRIPT_ACCEL*ACCEL_FACTOR, v=V_CIRC*SPEED_FACTOR, r=URSCRIPT_BLEND)
  movel(apply_correction(p[-0.020020, 0.568103, 0.050004, 3.141576, 0.000000, 0.000000]), a=URSCRIPT_ACCEL*ACCEL_FACTOR, v=V_CIRC*SPEED_FACTOR, r=URSCRIPT_BLEND)
  movel(apply_correction(p[-0.020718, 0.555702, 0.050005, 3.141576, 0.000000, 0.000000]), a=URSCRIPT_ACCEL*ACCEL_FACTOR, v=V_CIRC*SPEED_FACTOR, r=URSCRIPT_BLEND)
  movel(apply_correction(p[-0.008223, 0.555612, 0.050005, 3.141576, 0.000000, 0.000000]), a=URSCRIPT_ACCEL*ACCEL_FACTOR, v=V_CIRC*SPEED_FACTOR, r=URSCRIPT_BLEND)
  movel(apply_correction(p[-0.010804, 0.565438, 0.050004, 3.141576, 0.000000, 0.000000]), a=URSCRIPT_ACCEL*ACCEL_FACTOR, v=V_CIRC*SPEED_FACTOR, r=URSCRIPT_BLEND)
  movel(apply_correction(p[-0.019465, 0.558275, 0.050005, 3.141576, 0.000000, 0.000000]), a=URSCRIPT_ACCEL*ACCEL_FACTOR, v=V_CIRC*SPEED_FACTOR, r=URSCRIPT_BLEND)
  movel(apply_correction(p[-0.010180, 0.549212, 0.050005, 3.141576, 0.000000, 0.000000]), a=URSCRIPT_ACCEL*ACCEL_FACTOR, v=V_CIRC*SPEED_FACTOR, r=URSCRIPT_BLEND)
  movel(apply_correction(p[-0.003284, 0.558036, 0.050005, 3.141576, 0.000000, 0.000000]), a=URSCRIPT_ACCEL*ACCEL_FACTOR, v=V_CIRC*SPEED_FACTOR, r=URSCRIPT_BLEND)
  movel(apply_correction(p[-0.013205, 0.560317, 0.050005, 3.141576, 0.000000, 0.000000]), a=URSCRIPT_ACCEL*ACCEL_FACTOR, v=V_CIRC*SPEED_FACTOR, r=URSCRIPT_BLEND)
  movel(apply_correction(p[-0.012803, 0.547801, 0.050005, 3.141576, 0.000000, 0.000000]), a=URSCRIPT_ACCEL*ACCEL_FACTOR, v=V_CIRC*SPEED_FACTOR, r=URSCRIPT_BLEND)
  movel(apply_correction(p[-0.000454, 0.548808, 0.050005, 3.141576, 0.000000, 0.000000]), a=URSCRIPT_ACCEL*ACCEL_FACTOR, v=V_CIRC*SPEED_FACTOR, r=URSCRIPT_BLEND)
  movel(apply_correction(p[-0.001819, 0.552639, 0.050005, 3.141576, 0.000000, 0.000000]), a=URSCRIPT_ACCEL*ACCEL_FACTOR, v=V_CIRC*SPEED_FACTOR, r=URSCRIPT_BLEND)
  movel(apply_correction(p[-0.017675, 0.540361, 0.050005, 3.141576, 0.000000, 0.000000]), a=URSCRIPT_ACCEL*ACCEL_FACTOR, v=V_CIRC*SPEED_FACTOR, r=URSCRIPT_BLEND)
  movel(apply_correction(p[-0.021722, 0.540328, 0.050005, 3.141576, 0.000000, 0.000000]), a=URSCRIPT_ACCEL*ACCEL_FACTOR, v=V_CIRC*SPEED_FACTOR, r=URSCRIPT_BLEND)
  movel(apply_correction(p[-0.011399, 0.539911, 0.050005, 3.141576, 0.000000, 0.000000]), a=URSCRIPT_ACCEL*ACCEL_FACTOR, v=V_CIRC*SPEED_FACTOR, r=URSCRIPT_BLEND)
  movel(apply_correction(p[-0.013708, 0.552379, 0.050005, 3.141576, 0.000000, 0.000000]), a=URSCRIPT_ACCEL*ACCEL_FACTOR, v=V_CIRC*SPEED_FACTOR, r=URSCRIPT_BLEND)
  movel(apply_correction(p[-0.025558, 0.549529, 0.050005, 3.141576, 0.000000, 0.000000]), a=URSCRIPT_ACCEL*ACCEL_FACTOR, v=V_CIRC*SPEED_FACTOR, r=URSCRIPT_BLEND)
  movel(apply_correction(p[-0.020274, 0.541023, 0.050005, 3.141576, 0.000000, 0.000000]), a=URSCRIPT_ACCEL*ACCEL_FACTOR, v=V_CIRC*SPEED_FACTOR, r=URSCRIPT_BLEND)
  movel(apply_correction(p[-0.013534, 0.550503, 0.050005, 3.141576, 0.000000, 0.000000]), a=URSCRIPT_ACCEL*ACCEL_FACTOR, v=V_CIRC*SPEED_FACTOR, r=URSCRIPT_BLEND)
  movel(apply_correction(p[-0.024617, 0.557152, 0.050005, 3.141576, 0.000000, 0.000000]), a=URSCRIPT_ACCEL*ACCEL_FACTOR, v=V_CIRC*SPEED_FACTOR, r=URSCRIPT_BLEND)
  movel(apply_correction(p[-0.028743, 0.547152, 0.050005, 3.141576, 0.000000, 0.000000]), a=URSCRIPT_ACCEL*ACCEL_FACTOR, v=V_CIRC*SPEED_FACTOR, r=URSCRIPT_BLEND)
  movel(apply_correction(p[-0.018331, 0.547838, 0.050005, 3.141576, 0.000000, 0.000000]), a=URSCRIPT_ACCEL*ACCEL_FACTOR, v=V_CIRC*SPEED_FACTOR, r=URSCRIPT_BLEND)
  movel(apply_correction(p[-0.021734, 0.560131, 0.050005, 3.141576, 0.000000, 0.000000]), a=URSCRIPT_ACCEL*ACCEL_FACTOR, v=V_CIRC*SPEED_FACTOR, r=URSCRIPT_BLEND)
  movel(apply_correction(p[-0.033158, 0.556261, 0.050005, 3.141576, 0.000000, 0.000000]), a=URSCRIPT_ACCEL*ACCEL_FACTOR, v=V_CIRC*SPEED_FACTOR, r=URSCRIPT_BLEND)
  movel(apply_correction(p[-0.026980, 0.548411, 0.050005, 3.141576, 0.000000, 0.000000]), a=URSCRIPT_ACCEL*ACCEL_FACTOR, v=V_CIRC*SPEED_FACTOR, r=URSCRIPT_BLEND)
  movel(apply_correction(p[-0.021089, 0.558603, 0.050005, 3.141576, 0.000000, 0.000000]), a=URSCRIPT_ACCEL*ACCEL_FACTOR, v=V_CIRC*SPEED_FACTOR, r=URSCRIPT_BLEND)
  movel(apply_correction(p[-0.032663, 0.564261, 0.050005, 3.141576, 0.000000, 0.000000]), a=URSCRIPT_ACCEL*ACCEL_FACTOR, v=V_CIRC*SPEED_FACTOR, r=URSCRIPT_BLEND)
  movel(apply_correction(p[-0.035709, 0.554015, 0.050005, 3.141576, 0.000000, 0.000000]), a=URSCRIPT_ACCEL*ACCEL_FACTOR, v=V_CIRC*SPEED_FACTOR, r=URSCRIPT_BLEND)
  movel(apply_correction(p[-0.025315, 0.555810, 0.050005, 3.141576, 0.000000, 0.000000]), a=URSCRIPT_ACCEL*ACCEL_FACTOR, v=V_CIRC*SPEED_FACTOR, r=URSCRIPT_BLEND)
  movel(apply_correction(p[-0.029475, 0.567681, 0.050004, 3.141576, 0.000000, 0.000000]), a=URSCRIPT_ACCEL*ACCEL_FACTOR, v=V_CIRC*SPEED_FACTOR, r=URSCRIPT_BLEND)
  movel(apply_correction(p[-0.040636, 0.563198, 0.050005, 3.141576, 0.000000, 0.000000]), a=URSCRIPT_ACCEL*ACCEL_FACTOR, v=V_CIRC*SPEED_FACTOR, r=URSCRIPT_BLEND)
  movel(apply_correction(p[-0.033843, 0.555836, 0.050005, 3.141576, 0.000000, 0.000000]), a=URSCRIPT_ACCEL*ACCEL_FACTOR, v=V_CIRC*SPEED_FACTOR, r=URSCRIPT_BLEND)
  movel(apply_correction(p[-0.028668, 0.566586, 0.050004, 3.141576, 0.000000, 0.000000]), a=URSCRIPT_ACCEL*ACCEL_FACTOR, v=V_CIRC*SPEED_FACTOR, r=URSCRIPT_BLEND)
  movel(apply_correction(p[-0.040654, 0.571321, 0.050004, 3.141576, 0.000000, 0.000000]), a=URSCRIPT_ACCEL*ACCEL_FACTOR, v=V_CIRC*SPEED_FACTOR, r=URSCRIPT_BLEND)
  movel(apply_correction(p[-0.042820, 0.561110, 0.050005, 3.141576, 0.000000, 0.000000]), a=URSCRIPT_ACCEL*ACCEL_FACTOR, v=V_CIRC*SPEED_FACTOR, r=URSCRIPT_BLEND)
  end_force_mode()
  movel(apply_correction(p[-0.042820, 0.561110, 0.060005, 3.141576, 0.000000, 0.000000]), a=URSCRIPT_ACCEL*ACCEL_FACTOR, v=0.2500*SPEED_FACTOR)
end

def cycle_4():
  # --- Cycle 4 - Rectiligne (0deg) ---
  movel(apply_correction(p[-0.011000, 0.594344, 0.060004, 3.141576, 0.000000, 0.000000]), a=URSCRIPT_ACCEL*ACCEL_FACTOR, v=0.2500*SPEED_FACTOR)
  sleep(0.2)
  zero_ftsensor()
  sleep(0.2)
  force_mode(MEAS_FRAME, [0, 0, 1, 0, 0, 0], [0, 0, -6.0, 0, 0, 0], 2, [0.008, 0.008, 0.04, 0.35, 0.35, 0.35])
  movel(apply_correction(p[-0.011000, 0.594344, 0.045004, 3.141576, 0.000000, 0.000000]), a=URSCRIPT_ACCEL*ACCEL_FACTOR, v=URSCRIPT_RECONTACT_V*SPEED_FACTOR)
  movel(apply_correction(p[-0.011000, 0.594344, 0.050004, 3.141576, 0.000000, 0.000000]), a=URSCRIPT_ACCEL*ACCEL_FACTOR, v=V_RECT*SPEED_FACTOR, r=URSCRIPT_BLEND)
  movel(apply_correction(p[-0.040698, 0.564646, 0.050005, 3.141576, 0.000000, 0.000000]), a=URSCRIPT_ACCEL*ACCEL_FACTOR, v=V_RECT*SPEED_FACTOR, r=URSCRIPT_BLEND)
  movel(apply_correction(p[-0.038224, 0.562171, 0.050005, 3.141576, 0.000000, 0.000000]), a=URSCRIPT_ACCEL*ACCEL_FACTOR, v=V_RECT*SPEED_FACTOR, r=URSCRIPT_BLEND)
  movel(apply_correction(p[-0.008525, 0.591869, 0.050004, 3.141576, 0.000000, 0.000000]), a=URSCRIPT_ACCEL*ACCEL_FACTOR, v=V_RECT*SPEED_FACTOR, r=URSCRIPT_BLEND)
  movel(apply_correction(p[-0.006050, 0.589394, 0.050004, 3.141576, 0.000000, 0.000000]), a=URSCRIPT_ACCEL*ACCEL_FACTOR, v=V_RECT*SPEED_FACTOR, r=URSCRIPT_BLEND)
  movel(apply_correction(p[-0.035749, 0.559696, 0.050005, 3.141576, 0.000000, 0.000000]), a=URSCRIPT_ACCEL*ACCEL_FACTOR, v=V_RECT*SPEED_FACTOR, r=URSCRIPT_BLEND)
  movel(apply_correction(p[-0.033274, 0.557221, 0.050005, 3.141576, 0.000000, 0.000000]), a=URSCRIPT_ACCEL*ACCEL_FACTOR, v=V_RECT*SPEED_FACTOR, r=URSCRIPT_BLEND)
  movel(apply_correction(p[-0.003575, 0.586920, 0.050004, 3.141576, 0.000000, 0.000000]), a=URSCRIPT_ACCEL*ACCEL_FACTOR, v=V_RECT*SPEED_FACTOR, r=URSCRIPT_BLEND)
  movel(apply_correction(p[-0.001101, 0.584445, 0.050004, 3.141576, 0.000000, 0.000000]), a=URSCRIPT_ACCEL*ACCEL_FACTOR, v=V_RECT*SPEED_FACTOR, r=URSCRIPT_BLEND)
  movel(apply_correction(p[-0.030799, 0.554746, 0.050005, 3.141576, 0.000000, 0.000000]), a=URSCRIPT_ACCEL*ACCEL_FACTOR, v=V_RECT*SPEED_FACTOR, r=URSCRIPT_BLEND)
  movel(apply_correction(p[-0.028324, 0.552271, 0.050005, 3.141576, 0.000000, 0.000000]), a=URSCRIPT_ACCEL*ACCEL_FACTOR, v=V_RECT*SPEED_FACTOR, r=URSCRIPT_BLEND)
  movel(apply_correction(p[0.001374, 0.581970, 0.050004, 3.141576, 0.000000, 0.000000]), a=URSCRIPT_ACCEL*ACCEL_FACTOR, v=V_RECT*SPEED_FACTOR, r=URSCRIPT_BLEND)
  movel(apply_correction(p[0.003849, 0.579495, 0.050004, 3.141576, 0.000000, 0.000000]), a=URSCRIPT_ACCEL*ACCEL_FACTOR, v=V_RECT*SPEED_FACTOR, r=URSCRIPT_BLEND)
  movel(apply_correction(p[-0.025849, 0.549796, 0.050005, 3.141576, 0.000000, 0.000000]), a=URSCRIPT_ACCEL*ACCEL_FACTOR, v=V_RECT*SPEED_FACTOR, r=URSCRIPT_BLEND)
  movel(apply_correction(p[-0.023374, 0.547322, 0.050005, 3.141576, 0.000000, 0.000000]), a=URSCRIPT_ACCEL*ACCEL_FACTOR, v=V_RECT*SPEED_FACTOR, r=URSCRIPT_BLEND)
  movel(apply_correction(p[0.006324, 0.577020, 0.050004, 3.141576, 0.000000, 0.000000]), a=URSCRIPT_ACCEL*ACCEL_FACTOR, v=V_RECT*SPEED_FACTOR, r=URSCRIPT_BLEND)
  movel(apply_correction(p[0.008799, 0.574545, 0.050004, 3.141576, 0.000000, 0.000000]), a=URSCRIPT_ACCEL*ACCEL_FACTOR, v=V_RECT*SPEED_FACTOR, r=URSCRIPT_BLEND)
  movel(apply_correction(p[-0.020899, 0.544847, 0.050005, 3.141576, 0.000000, 0.000000]), a=URSCRIPT_ACCEL*ACCEL_FACTOR, v=V_RECT*SPEED_FACTOR, r=URSCRIPT_BLEND)
  movel(apply_correction(p[-0.018425, 0.542372, 0.050005, 3.141576, 0.000000, 0.000000]), a=URSCRIPT_ACCEL*ACCEL_FACTOR, v=V_RECT*SPEED_FACTOR, r=URSCRIPT_BLEND)
  movel(apply_correction(p[0.011274, 0.572070, 0.050004, 3.141576, 0.000000, 0.000000]), a=URSCRIPT_ACCEL*ACCEL_FACTOR, v=V_RECT*SPEED_FACTOR, r=URSCRIPT_BLEND)
  movel(apply_correction(p[0.013749, 0.569595, 0.050004, 3.141576, 0.000000, 0.000000]), a=URSCRIPT_ACCEL*ACCEL_FACTOR, v=V_RECT*SPEED_FACTOR, r=URSCRIPT_BLEND)
  movel(apply_correction(p[-0.015950, 0.539897, 0.050005, 3.141576, 0.000000, 0.000000]), a=URSCRIPT_ACCEL*ACCEL_FACTOR, v=V_RECT*SPEED_FACTOR, r=URSCRIPT_BLEND)
  movel(apply_correction(p[-0.013475, 0.537422, 0.050005, 3.141576, 0.000000, 0.000000]), a=URSCRIPT_ACCEL*ACCEL_FACTOR, v=V_RECT*SPEED_FACTOR, r=URSCRIPT_BLEND)
  movel(apply_correction(p[0.016224, 0.567121, 0.050004, 3.141576, 0.000000, 0.000000]), a=URSCRIPT_ACCEL*ACCEL_FACTOR, v=V_RECT*SPEED_FACTOR, r=URSCRIPT_BLEND)
  movel(apply_correction(p[0.018698, 0.564646, 0.050005, 3.141576, 0.000000, 0.000000]), a=URSCRIPT_ACCEL*ACCEL_FACTOR, v=V_RECT*SPEED_FACTOR, r=URSCRIPT_BLEND)
  movel(apply_correction(p[-0.011000, 0.534947, 0.050005, 3.141576, 0.000000, 0.000000]), a=URSCRIPT_ACCEL*ACCEL_FACTOR, v=V_RECT*SPEED_FACTOR, r=URSCRIPT_BLEND)
  end_force_mode()
  movel(apply_correction(p[-0.011000, 0.534947, 0.060005, 3.141576, 0.000000, 0.000000]), a=URSCRIPT_ACCEL*ACCEL_FACTOR, v=0.2500*SPEED_FACTOR)
end

def cycle_5():
  # --- Cycle 5 - Rectiligne (90deg) ---
  movel(apply_correction(p[-0.040698, 0.564646, 0.060005, 3.141576, 0.000000, 0.000000]), a=URSCRIPT_ACCEL*ACCEL_FACTOR, v=0.2500*SPEED_FACTOR)
  sleep(0.2)
  zero_ftsensor()
  sleep(0.2)
  force_mode(MEAS_FRAME, [0, 0, 1, 0, 0, 0], [0, 0, -6.0, 0, 0, 0], 2, [0.008, 0.008, 0.04, 0.35, 0.35, 0.35])
  movel(apply_correction(p[-0.040698, 0.564646, 0.045005, 3.141576, 0.000000, 0.000000]), a=URSCRIPT_ACCEL*ACCEL_FACTOR, v=URSCRIPT_RECONTACT_V*SPEED_FACTOR)
  movel(apply_correction(p[-0.040698, 0.564646, 0.050005, 3.141576, 0.000000, 0.000000]), a=URSCRIPT_ACCEL*ACCEL_FACTOR, v=V_RECT*SPEED_FACTOR, r=URSCRIPT_BLEND)
  movel(apply_correction(p[-0.011000, 0.534947, 0.050005, 3.141576, 0.000000, 0.000000]), a=URSCRIPT_ACCEL*ACCEL_FACTOR, v=V_RECT*SPEED_FACTOR, r=URSCRIPT_BLEND)
  movel(apply_correction(p[-0.008525, 0.537422, 0.050005, 3.141576, 0.000000, 0.000000]), a=URSCRIPT_ACCEL*ACCEL_FACTOR, v=V_RECT*SPEED_FACTOR, r=URSCRIPT_BLEND)
  movel(apply_correction(p[-0.038224, 0.567121, 0.050004, 3.141576, 0.000000, 0.000000]), a=URSCRIPT_ACCEL*ACCEL_FACTOR, v=V_RECT*SPEED_FACTOR, r=URSCRIPT_BLEND)
  movel(apply_correction(p[-0.035749, 0.569595, 0.050004, 3.141576, 0.000000, 0.000000]), a=URSCRIPT_ACCEL*ACCEL_FACTOR, v=V_RECT*SPEED_FACTOR, r=URSCRIPT_BLEND)
  movel(apply_correction(p[-0.006050, 0.539897, 0.050005, 3.141576, 0.000000, 0.000000]), a=URSCRIPT_ACCEL*ACCEL_FACTOR, v=V_RECT*SPEED_FACTOR, r=URSCRIPT_BLEND)
  movel(apply_correction(p[-0.003575, 0.542372, 0.050005, 3.141576, 0.000000, 0.000000]), a=URSCRIPT_ACCEL*ACCEL_FACTOR, v=V_RECT*SPEED_FACTOR, r=URSCRIPT_BLEND)
  movel(apply_correction(p[-0.033274, 0.572070, 0.050004, 3.141576, 0.000000, 0.000000]), a=URSCRIPT_ACCEL*ACCEL_FACTOR, v=V_RECT*SPEED_FACTOR, r=URSCRIPT_BLEND)
  movel(apply_correction(p[-0.030799, 0.574545, 0.050004, 3.141576, 0.000000, 0.000000]), a=URSCRIPT_ACCEL*ACCEL_FACTOR, v=V_RECT*SPEED_FACTOR, r=URSCRIPT_BLEND)
  movel(apply_correction(p[-0.001101, 0.544847, 0.050005, 3.141576, 0.000000, 0.000000]), a=URSCRIPT_ACCEL*ACCEL_FACTOR, v=V_RECT*SPEED_FACTOR, r=URSCRIPT_BLEND)
  movel(apply_correction(p[0.001374, 0.547322, 0.050005, 3.141576, 0.000000, 0.000000]), a=URSCRIPT_ACCEL*ACCEL_FACTOR, v=V_RECT*SPEED_FACTOR, r=URSCRIPT_BLEND)
  movel(apply_correction(p[-0.028324, 0.577020, 0.050004, 3.141576, 0.000000, 0.000000]), a=URSCRIPT_ACCEL*ACCEL_FACTOR, v=V_RECT*SPEED_FACTOR, r=URSCRIPT_BLEND)
  movel(apply_correction(p[-0.025849, 0.579495, 0.050004, 3.141576, 0.000000, 0.000000]), a=URSCRIPT_ACCEL*ACCEL_FACTOR, v=V_RECT*SPEED_FACTOR, r=URSCRIPT_BLEND)
  movel(apply_correction(p[0.003849, 0.549796, 0.050005, 3.141576, 0.000000, 0.000000]), a=URSCRIPT_ACCEL*ACCEL_FACTOR, v=V_RECT*SPEED_FACTOR, r=URSCRIPT_BLEND)
  movel(apply_correction(p[0.006324, 0.552271, 0.050005, 3.141576, 0.000000, 0.000000]), a=URSCRIPT_ACCEL*ACCEL_FACTOR, v=V_RECT*SPEED_FACTOR, r=URSCRIPT_BLEND)
  movel(apply_correction(p[-0.023374, 0.581970, 0.050004, 3.141576, 0.000000, 0.000000]), a=URSCRIPT_ACCEL*ACCEL_FACTOR, v=V_RECT*SPEED_FACTOR, r=URSCRIPT_BLEND)
  movel(apply_correction(p[-0.020899, 0.584445, 0.050004, 3.141576, 0.000000, 0.000000]), a=URSCRIPT_ACCEL*ACCEL_FACTOR, v=V_RECT*SPEED_FACTOR, r=URSCRIPT_BLEND)
  movel(apply_correction(p[0.008799, 0.554746, 0.050005, 3.141576, 0.000000, 0.000000]), a=URSCRIPT_ACCEL*ACCEL_FACTOR, v=V_RECT*SPEED_FACTOR, r=URSCRIPT_BLEND)
  movel(apply_correction(p[0.011274, 0.557221, 0.050005, 3.141576, 0.000000, 0.000000]), a=URSCRIPT_ACCEL*ACCEL_FACTOR, v=V_RECT*SPEED_FACTOR, r=URSCRIPT_BLEND)
  movel(apply_correction(p[-0.018425, 0.586920, 0.050004, 3.141576, 0.000000, 0.000000]), a=URSCRIPT_ACCEL*ACCEL_FACTOR, v=V_RECT*SPEED_FACTOR, r=URSCRIPT_BLEND)
  movel(apply_correction(p[-0.015950, 0.589394, 0.050004, 3.141576, 0.000000, 0.000000]), a=URSCRIPT_ACCEL*ACCEL_FACTOR, v=V_RECT*SPEED_FACTOR, r=URSCRIPT_BLEND)
  movel(apply_correction(p[0.013749, 0.559696, 0.050005, 3.141576, 0.000000, 0.000000]), a=URSCRIPT_ACCEL*ACCEL_FACTOR, v=V_RECT*SPEED_FACTOR, r=URSCRIPT_BLEND)
  movel(apply_correction(p[0.016224, 0.562171, 0.050005, 3.141576, 0.000000, 0.000000]), a=URSCRIPT_ACCEL*ACCEL_FACTOR, v=V_RECT*SPEED_FACTOR, r=URSCRIPT_BLEND)
  movel(apply_correction(p[-0.013475, 0.591869, 0.050004, 3.141576, 0.000000, 0.000000]), a=URSCRIPT_ACCEL*ACCEL_FACTOR, v=V_RECT*SPEED_FACTOR, r=URSCRIPT_BLEND)
  movel(apply_correction(p[-0.011000, 0.594344, 0.050004, 3.141576, 0.000000, 0.000000]), a=URSCRIPT_ACCEL*ACCEL_FACTOR, v=V_RECT*SPEED_FACTOR, r=URSCRIPT_BLEND)
  movel(apply_correction(p[0.018698, 0.564646, 0.050005, 3.141576, 0.000000, 0.000000]), a=URSCRIPT_ACCEL*ACCEL_FACTOR, v=V_RECT*SPEED_FACTOR, r=URSCRIPT_BLEND)
  end_force_mode()
  movel(apply_correction(p[0.018698, 0.564646, 0.060005, 3.141576, 0.000000, 0.000000]), a=URSCRIPT_ACCEL*ACCEL_FACTOR, v=0.2500*SPEED_FACTOR)
end

def cycle_6():
  # --- Cycle 6 - Rectiligne (0deg) ---
  movel(apply_correction(p[-0.011000, 0.594344, 0.060004, 3.141576, 0.000000, 0.000000]), a=URSCRIPT_ACCEL*ACCEL_FACTOR, v=0.2500*SPEED_FACTOR)
  sleep(0.2)
  zero_ftsensor()
  sleep(0.2)
  force_mode(MEAS_FRAME, [0, 0, 1, 0, 0, 0], [0, 0, -6.0, 0, 0, 0], 2, [0.008, 0.008, 0.04, 0.35, 0.35, 0.35])
  movel(apply_correction(p[-0.011000, 0.594344, 0.045004, 3.141576, 0.000000, 0.000000]), a=URSCRIPT_ACCEL*ACCEL_FACTOR, v=URSCRIPT_RECONTACT_V*SPEED_FACTOR)
  movel(apply_correction(p[-0.011000, 0.594344, 0.050004, 3.141576, 0.000000, 0.000000]), a=URSCRIPT_ACCEL*ACCEL_FACTOR, v=V_RECT*SPEED_FACTOR, r=URSCRIPT_BLEND)
  movel(apply_correction(p[-0.040698, 0.564646, 0.050005, 3.141576, 0.000000, 0.000000]), a=URSCRIPT_ACCEL*ACCEL_FACTOR, v=V_RECT*SPEED_FACTOR, r=URSCRIPT_BLEND)
  movel(apply_correction(p[-0.038224, 0.562171, 0.050005, 3.141576, 0.000000, 0.000000]), a=URSCRIPT_ACCEL*ACCEL_FACTOR, v=V_RECT*SPEED_FACTOR, r=URSCRIPT_BLEND)
  movel(apply_correction(p[-0.008525, 0.591869, 0.050004, 3.141576, 0.000000, 0.000000]), a=URSCRIPT_ACCEL*ACCEL_FACTOR, v=V_RECT*SPEED_FACTOR, r=URSCRIPT_BLEND)
  movel(apply_correction(p[-0.006050, 0.589394, 0.050004, 3.141576, 0.000000, 0.000000]), a=URSCRIPT_ACCEL*ACCEL_FACTOR, v=V_RECT*SPEED_FACTOR, r=URSCRIPT_BLEND)
  movel(apply_correction(p[-0.035749, 0.559696, 0.050005, 3.141576, 0.000000, 0.000000]), a=URSCRIPT_ACCEL*ACCEL_FACTOR, v=V_RECT*SPEED_FACTOR, r=URSCRIPT_BLEND)
  movel(apply_correction(p[-0.033274, 0.557221, 0.050005, 3.141576, 0.000000, 0.000000]), a=URSCRIPT_ACCEL*ACCEL_FACTOR, v=V_RECT*SPEED_FACTOR, r=URSCRIPT_BLEND)
  movel(apply_correction(p[-0.003575, 0.586920, 0.050004, 3.141576, 0.000000, 0.000000]), a=URSCRIPT_ACCEL*ACCEL_FACTOR, v=V_RECT*SPEED_FACTOR, r=URSCRIPT_BLEND)
  movel(apply_correction(p[-0.001101, 0.584445, 0.050004, 3.141576, 0.000000, 0.000000]), a=URSCRIPT_ACCEL*ACCEL_FACTOR, v=V_RECT*SPEED_FACTOR, r=URSCRIPT_BLEND)
  movel(apply_correction(p[-0.030799, 0.554746, 0.050005, 3.141576, 0.000000, 0.000000]), a=URSCRIPT_ACCEL*ACCEL_FACTOR, v=V_RECT*SPEED_FACTOR, r=URSCRIPT_BLEND)
  movel(apply_correction(p[-0.028324, 0.552271, 0.050005, 3.141576, 0.000000, 0.000000]), a=URSCRIPT_ACCEL*ACCEL_FACTOR, v=V_RECT*SPEED_FACTOR, r=URSCRIPT_BLEND)
  movel(apply_correction(p[0.001374, 0.581970, 0.050004, 3.141576, 0.000000, 0.000000]), a=URSCRIPT_ACCEL*ACCEL_FACTOR, v=V_RECT*SPEED_FACTOR, r=URSCRIPT_BLEND)
  movel(apply_correction(p[0.003849, 0.579495, 0.050004, 3.141576, 0.000000, 0.000000]), a=URSCRIPT_ACCEL*ACCEL_FACTOR, v=V_RECT*SPEED_FACTOR, r=URSCRIPT_BLEND)
  movel(apply_correction(p[-0.025849, 0.549796, 0.050005, 3.141576, 0.000000, 0.000000]), a=URSCRIPT_ACCEL*ACCEL_FACTOR, v=V_RECT*SPEED_FACTOR, r=URSCRIPT_BLEND)
  movel(apply_correction(p[-0.023374, 0.547322, 0.050005, 3.141576, 0.000000, 0.000000]), a=URSCRIPT_ACCEL*ACCEL_FACTOR, v=V_RECT*SPEED_FACTOR, r=URSCRIPT_BLEND)
  movel(apply_correction(p[0.006324, 0.577020, 0.050004, 3.141576, 0.000000, 0.000000]), a=URSCRIPT_ACCEL*ACCEL_FACTOR, v=V_RECT*SPEED_FACTOR, r=URSCRIPT_BLEND)
  movel(apply_correction(p[0.008799, 0.574545, 0.050004, 3.141576, 0.000000, 0.000000]), a=URSCRIPT_ACCEL*ACCEL_FACTOR, v=V_RECT*SPEED_FACTOR, r=URSCRIPT_BLEND)
  movel(apply_correction(p[-0.020899, 0.544847, 0.050005, 3.141576, 0.000000, 0.000000]), a=URSCRIPT_ACCEL*ACCEL_FACTOR, v=V_RECT*SPEED_FACTOR, r=URSCRIPT_BLEND)
  movel(apply_correction(p[-0.018425, 0.542372, 0.050005, 3.141576, 0.000000, 0.000000]), a=URSCRIPT_ACCEL*ACCEL_FACTOR, v=V_RECT*SPEED_FACTOR, r=URSCRIPT_BLEND)
  movel(apply_correction(p[0.011274, 0.572070, 0.050004, 3.141576, 0.000000, 0.000000]), a=URSCRIPT_ACCEL*ACCEL_FACTOR, v=V_RECT*SPEED_FACTOR, r=URSCRIPT_BLEND)
  movel(apply_correction(p[0.013749, 0.569595, 0.050004, 3.141576, 0.000000, 0.000000]), a=URSCRIPT_ACCEL*ACCEL_FACTOR, v=V_RECT*SPEED_FACTOR, r=URSCRIPT_BLEND)
  movel(apply_correction(p[-0.015950, 0.539897, 0.050005, 3.141576, 0.000000, 0.000000]), a=URSCRIPT_ACCEL*ACCEL_FACTOR, v=V_RECT*SPEED_FACTOR, r=URSCRIPT_BLEND)
  movel(apply_correction(p[-0.013475, 0.537422, 0.050005, 3.141576, 0.000000, 0.000000]), a=URSCRIPT_ACCEL*ACCEL_FACTOR, v=V_RECT*SPEED_FACTOR, r=URSCRIPT_BLEND)
  movel(apply_correction(p[0.016224, 0.567121, 0.050004, 3.141576, 0.000000, 0.000000]), a=URSCRIPT_ACCEL*ACCEL_FACTOR, v=V_RECT*SPEED_FACTOR, r=URSCRIPT_BLEND)
  movel(apply_correction(p[0.018698, 0.564646, 0.050005, 3.141576, 0.000000, 0.000000]), a=URSCRIPT_ACCEL*ACCEL_FACTOR, v=V_RECT*SPEED_FACTOR, r=URSCRIPT_BLEND)
  movel(apply_correction(p[-0.011000, 0.534947, 0.050005, 3.141576, 0.000000, 0.000000]), a=URSCRIPT_ACCEL*ACCEL_FACTOR, v=V_RECT*SPEED_FACTOR, r=URSCRIPT_BLEND)
  end_force_mode()
  movel(apply_correction(p[-0.011000, 0.534947, 0.060005, 3.141576, 0.000000, 0.000000]), a=URSCRIPT_ACCEL*ACCEL_FACTOR, v=0.2500*SPEED_FACTOR)
end

def etalement():
  set_tcp(p[0.0, 0.0, 0.2657, 0, 0, 0])
  # Aucune pose home absolue : la position de depart est la pose courante
  # du robot (mesuree a l'execution). L'operateur jogge le robot ou il
  # veut, clique Start, et le sondage de surface part de la.
  home = get_actual_tcp_pose()
  probe_surface_z()

  cycle_1()
  cycle_2()
  cycle_3()
  cycle_4()
  cycle_5()
  cycle_6()
  movel(apply_correction(p[-0.011000, 0.534947, 0.080005, 3.141576, 0.000000, 0.000000]), a=URSCRIPT_ACCEL*ACCEL_FACTOR, v=0.2500*SPEED_FACTOR)
end

etalement()
